  MoveL 4062 to (-40.22, 47.43, 69.25) mm, rotated rx 180 ry 0 rz -180 deg; joints [-39.002, -24.615, 92.109, 64.701, 44.116, -56.64]
  Call Extruder(62.49416)
  MoveL 4063 to (-40.17, 47.23, 69.25) mm, rotated rx 180 ry 0 rz 180 deg; joints [-38.962, -24.627, 92.115, 64.664, 44.084, -56.61]
  MoveL 4064 to (-40.17, 47.23, 69.25) mm, rotated rx 180 ry 0 rz 180 deg; joints [-38.962, -24.627, 92.115, 64.664, 44.084, -56.61]
  Call Extruder(62.60834)
  MoveL 4065 to (-40.13, 47.02, 69.25) mm, rotated rx 180 ry 0 rz 180 deg; joints [-38.921, -24.64, 92.122, 64.627, 44.053, -56.579]
  MoveL 4066 to (-40.13, 47.02, 69.25) mm, rotated rx 180 ry 0 rz 180 deg; joints [-38.921, -24.64, 92.122, 64.627, 44.053, -56.579]
  Call Extruder(62.72297)
  MoveL 4067 to (-40.08, 46.82, 69.25) mm, rotated rx 180 ry 0 rz -180 deg; joints [-38.88, -24.652, 92.129, 64.589, 44.021, -56.549]
  MoveL 4068 to (-40.08, 46.82, 69.25) mm, rotated rx 180 ry 0 rz -180 deg; joints [-38.88, -24.652, 92.129, 64.589, 44.021, -56.549]
  Call Extruder(62.83806)
  MoveL 4069 to (-40.04, 46.61, 69.25) mm, rotated rx 180 ry 0 rz 180 deg; joints [-38.839, -24.664, 92.136, 64.552, 43.989, -56.519]
  MoveL 4070 to (-40.04, 46.61, 69.25) mm, rotated rx 180 ry 0 rz 180 deg; joints [-38.839, -24.664, 92.136, 64.552, 43.989, -56.519]
  Call Extruder(62.96029)
  MoveL 4071 to (-39.98, 46.4, 69.25) mm, rotated rx 180 ry 0 rz 180 deg; joints [-38.795, -24.676, 92.142, 64.512, 43.955, -56.487]
  MoveL 4072 to (-39.98, 46.4, 69.25) mm, rotated rx 180 ry 0 rz 180 deg; joints [-38.795, -24.676, 92.142, 64.512, 43.955, -56.487]
  Call Extruder(63.08996)
  MoveL 4073 to (-39.92, 46.18, 69.25) mm, rotated rx 180 ry 0 rz -180 deg; joints [-38.748, -24.687, 92.148, 64.469, 43.917, -56.453]
  MoveL 4074 to (-39.92, 46.18, 69.25) mm, rotated rx 180 ry 0 rz -180 deg; joints [-38.748, -24.687, 92.148, 64.469, 43.917, -56.453]
  Call Extruder(63.22019)
  MoveL 4075 to (-39.85, 45.95, 69.25) mm, rotated rx 180 ry 0 rz 180 deg; joints [-38.7, -24.699, 92.155, 64.427, 43.88, -56.419]
  MoveL 4076 to (-39.85, 45.95, 69.25) mm, rotated rx 180 ry 0 rz 180 deg; joints [-38.7, -24.699, 92.155, 64.427, 43.88, -56.419]
  Call Extruder(63.35098)
  MoveL 4077 to (-39.78, 45.73, 69.25) mm, rotated rx 180 ry 0 rz 180 deg; joints [-38.653, -24.71, 92.161, 64.384, 43.843, -56.385]
  MoveL 4078 to (-39.78, 45.73, 69.25) mm, rotated rx 180 ry 0 rz 180 deg; joints [-38.653, -24.71, 92.161, 64.384, 43.843, -56.385]
  Call Extruder(63.48234)
  MoveL 4079 to (-39.71, 45.51, 69.25) mm, rotated rx 180 ry 0 rz 180 deg; joints [-38.605, -24.721, 92.167, 64.341, 43.805, -56.351]
  MoveL 4080 to (-39.71, 45.51, 69.25) mm, rotated rx 180 ry 0 rz 180 deg; joints [-38.605, -24.721, 92.167, 64.341, 43.805, -56.351]
  Call Extruder(63.59424)
  MoveL 4081 to (-39.65, 45.32, 69.25) mm, rotated rx -180 ry 0 rz 180 deg; joints [-38.565, -24.73, 92.172, 64.305, 43.774, -56.322]
  MoveL 4082 to (-39.65, 45.32, 69.25) mm, rotated rx -180 ry 0 rz 180 deg; joints [-38.565, -24.73, 92.172, 64.305, 43.774, -56.322]
  Call Extruder(63.70659)
  MoveL 4083 to (-39.59, 45.13, 69.25) mm, rotated rx 180 ry 0 rz 180 deg; joints [-38.524, -24.74, 92.177, 64.268, 43.741, -56.293]
  MoveL 4084 to (-39.59, 45.13, 69.25) mm, rotated rx 180 ry 0 rz 180 deg; joints [-38.524, -24.74, 92.177, 64.268, 43.741, -56.293]
  Call Extruder(63.81938)
  MoveL 4085 to (-39.53, 44.94, 69.25) mm, rotated rx 180 ry 0 rz -180 deg; joints [-38.483, -24.749, 92.182, 64.232, 43.709, -56.264]
  MoveL 4086 to (-39.53, 44.94, 69.25) mm, rotated rx 180 ry 0 rz -180 deg; joints [-38.483, -24.749, 92.182, 64.232, 43.709, -56.264]
  Call Extruder(63.93261)
  MoveL 4087 to (-39.47, 44.75, 69.25) mm, rotated rx -180 ry 0 rz 180 deg; joints [-38.443, -24.758, 92.187, 64.195, 43.677, -56.235]
  MoveL 4088 to (-39.47, 44.75, 69.25) mm, rotated rx -180 ry 0 rz 180 deg; joints [-38.443, -24.758, 92.187, 64.195, 43.677, -56.235]
  Call Extruder(64.04629)
  MoveL 4089 to (-39.41, 44.56, 69.25) mm, rotated rx -180 ry 0 rz 180 deg; joints [-38.402, -24.767, 92.192, 64.159, 43.645, -56.206]
  MoveL 4090 to (-39.41, 44.56, 69.25) mm, rotated rx -180 ry 0 rz 180 deg; joints [-38.402, -24.767, 92.192, 64.159, 43.645, -56.206]
  Call Extruder(64.22825)
  MoveL 4091 to (-39.29, 44.27, 69.25) mm, rotated rx 180 ry 0 rz 180 deg; joints [-38.335, -24.778, 92.198, 64.1, 43.592, -56.161]
  MoveL 4092 to (-39.29, 44.27, 69.25) mm, rotated rx 180 ry 0 rz 180 deg; joints [-38.335, -24.778, 92.198, 64.1, 43.592, -56.161]
  Call Extruder(64.41097)
  MoveL 4093 to (-39.16, 43.98, 69.25) mm, rotated rx -180 ry 0 rz 180 deg; joints [-38.269, -24.789, 92.204, 64.042, 43.539, -56.115]
  MoveL 4094 to (-39.16, 43.98, 69.25) mm, rotated rx -180 ry 0 rz 180 deg; joints [-38.269, -24.789, 92.204, 64.042, 43.539, -56.115]
  Call Extruder(64.58138)
  MoveL 4095 to (-39.05, 43.71, 69.25) mm, rotated rx 180 ry 0 rz 180 deg; joints [-38.207, -24.799, 92.21, 63.987, 43.49, -56.073]
  MoveL 4096 to (-39.05, 43.71, 69.25) mm, rotated rx 180 ry 0 rz 180 deg; joints [-38.207, -24.799, 92.21, 63.987, 43.49, -56.073]
  Call Extruder(64.73937)
  MoveL 4097 to (-38.94, 43.46, 69.25) mm, rotated rx 180 ry 0 rz 180 deg; joints [-38.149, -24.808, 92.215, 63.936, 43.444, -56.034]
  MoveL 4098 to (-38.94, 43.46, 69.25) mm, rotated rx 180 ry 0 rz 180 deg; joints [-38.149, -24.808, 92.215, 63.936, 43.444, -56.034]
  Call Extruder(64.89795)
  MoveL 4099 to (-38.84, 43.21, 69.25) mm, rotated rx 180 ry 0 rz 180 deg; joints [-38.092, -24.818, 92.22, 63.886, 43.398, -55.994]
  MoveL 4100 to (-38.84, 43.21, 69.25) mm, rotated rx 180 ry 0 rz 180 deg; joints [-38.092, -24.818, 92.22, 63.886, 43.398, -55.994]
  Call Extruder(65.10412)
  MoveL 4101 to (-38.66, 42.91, 69.25) mm, rotated rx 180 ry 0 rz 180 deg; joints [-38.016, -24.824, 92.224, 63.821, 43.336, -55.945]
  MoveL 4102 to (-38.66, 42.91, 69.25) mm, rotated rx 180 ry 0 rz 180 deg; joints [-38.016, -24.824, 92.224, 63.821, 43.336, -55.945]
  Call Extruder(65.31106)
  MoveL 4103 to (-38.49, 42.6, 69.25) mm, rotated rx 180 ry 0 rz -180 deg; joints [-37.939, -24.83, 92.227, 63.756, 43.274, -55.896]
  MoveL 4104 to (-38.49, 42.6, 69.25) mm, rotated rx 180 ry 0 rz -180 deg; joints [-37.939, -24.83, 92.227, 63.756, 43.274, -55.896]
  Call Extruder(65.51879)
  MoveL 4105 to (-38.31, 42.3, 69.25) mm, rotated rx -180 ry 0 rz 180 deg; joints [-37.863, -24.837, 92.23, 63.69, 43.212, -55.847]
  MoveL 4106 to (-38.31, 42.3, 69.25) mm, rotated rx -180 ry 0 rz 180 deg; joints [-37.863, -24.837, 92.23, 63.69, 43.212, -55.847]
  Call Extruder(65.72729)
  MoveL 4107 to (-38.14, 41.99, 69.25) mm, rotated rx 180 ry 0 rz 180 deg; joints [-37.787, -24.843, 92.234, 63.625, 43.15, -55.797]
  MoveL 4108 to (-38.14, 41.99, 69.25) mm, rotated rx 180 ry 0 rz 180 deg; joints [-37.787, -24.843, 92.234, 63.625, 43.15, -55.797]
  Call Extruder(65.90684)
  MoveL 4109 to (-37.96, 41.75, 69.25) mm, rotated rx -180 ry 0 rz 180 deg; joints [-37.72, -24.844, 92.235, 63.57, 43.096, -55.757]
  MoveL 4110 to (-37.96, 41.75, 69.25) mm, rotated rx -180 ry 0 rz 180 deg; joints [-37.72, -24.844, 92.235, 63.57, 43.096, -55.757]
  Call Extruder(66.24028)
  MoveL 4111 to (-37.63, 41.3, 69.25) mm, rotated rx 180 ry 0 rz -180 deg; joints [-37.598, -24.846, 92.236, 63.468, 42.995, -55.682]
  MoveL 4112 to (-37.63, 41.3, 69.25) mm, rotated rx 180 ry 0 rz -180 deg; joints [-37.598, -24.846, 92.236, 63.468, 42.995, -55.682]
  Call Extruder(66.57490)
  MoveL 4113 to (-37.3, 40.85, 69.25) mm, rotated rx 180 ry 0 rz 180 deg; joints [-37.475, -24.848, 92.237, 63.366, 42.894, -55.606]
  Call Extruder(67.40283)
  MoveL 4114 to (-36.39, 39.81, 69.25) mm, rotated rx -180 ry 0 rz 180 deg; joints [-37.173, -24.836, 92.23, 63.119, 42.642, -55.429]
  Call Extruder(68.23074)
  MoveL 4115 to (-35.35, 38.9, 69.25) mm, rotated rx 180 ry 0 rz 180 deg; joints [-36.876, -24.799, 92.21, 62.885, 42.391, -55.266]
  Call Extruder(68.39804)
  MoveL 4116 to (-35.13, 38.73, 69.25) mm, rotated rx -180 ry 0 rz -180 deg; joints [-36.818, -24.789, 92.204, 62.84, 42.34, -55.236]
  MoveL 4117 to (-35.13, 38.73, 69.25) mm, rotated rx -180 ry 0 rz -180 deg; joints [-36.818, -24.789, 92.204, 62.84, 42.34, -55.236]
  Call Extruder(68.73147)
  MoveL 4118 to (-34.68, 38.41, 69.25) mm, rotated rx 180 ry 0 rz 180 deg; joints [-36.701, -24.767, 92.192, 62.751, 42.24, -55.176]
  MoveL 4119 to (-34.68, 38.41, 69.25) mm, rotated rx 180 ry 0 rz 180 deg; joints [-36.701, -24.767, 92.192, 62.751, 42.24, -55.176]
  Call Extruder(69.06371)
  MoveL 4120 to (-34.23, 38.08, 69.25) mm, rotated rx 180 ry 0 rz -180 deg; joints [-36.584, -24.745, 92.18, 62.661, 42.14, -55.115]
  MoveL 4121 to (-34.23, 38.08, 69.25) mm, rotated rx 180 ry 0 rz -180 deg; joints [-36.584, -24.745, 92.18, 62.661, 42.14, -55.115]
  Call Extruder(69.18141)
  MoveL 4122 to (-34.05, 37.98, 69.25) mm, rotated rx 180 ry 0 rz 180 deg; joints [-36.544, -24.735, 92.175, 62.632, 42.105, -55.096]
  MoveL 4123 to (-34.05, 37.98, 69.25) mm, rotated rx 180 ry 0 rz 180 deg; joints [-36.544, -24.735, 92.175, 62.632, 42.105, -55.096]
  Call Extruder(69.38913)
  MoveL 4124 to (-33.75, 37.8, 69.25) mm, rotated rx 180 ry 0 rz 180 deg; joints [-36.474, -24.717, 92.165, 62.58, 42.043, -55.062]
  MoveL 4125 to (-33.75, 37.8, 69.25) mm, rotated rx 180 ry 0 rz 180 deg; joints [-36.474, -24.717, 92.165, 62.58, 42.043, -55.062]
  Call Extruder(69.59607)
  MoveL 4126 to (-33.45, 37.63, 69.25) mm, rotated rx 180 ry 0 rz 180 deg; joints [-36.403, -24.699, 92.155, 62.527, 41.982, -55.028]
  MoveL 4127 to (-33.45, 37.63, 69.25) mm, rotated rx 180 ry 0 rz 180 deg; joints [-36.403, -24.699, 92.155, 62.527, 41.982, -55.028]
  Call Extruder(69.80224)
  MoveL 4128 to (-33.14, 37.45, 69.25) mm, rotated rx 180 ry 0 rz 180 deg; joints [-36.333, -24.68, 92.144, 62.475, 41.921, -54.994]
  MoveL 4129 to (-33.14, 37.45, 69.25) mm, rotated rx 180 ry 0 rz 180 deg; joints [-36.333, -24.68, 92.144, 62.475, 41.921, -54.994]
  Call Extruder(69.98392)
  MoveL 4130 to (-32.86, 37.31, 69.25) mm, rotated rx 180 ry 0 rz 180 deg; joints [-36.272, -24.662, 92.134, 62.431, 41.867, -54.966]
  MoveL 4131 to (-32.86, 37.31, 69.25) mm, rotated rx 180 ry 0 rz 180 deg; joints [-36.272, -24.662, 92.134, 62.431, 41.867, -54.966]
  Call Extruder(70.14192)
  MoveL 4132 to (-32.62, 37.2, 69.25) mm, rotated rx 180 ry 0 rz 180 deg; joints [-36.221, -24.644, 92.124, 62.395, 41.822, -54.944]
  MoveL 4133 to (-32.62, 37.2, 69.25) mm, rotated rx 180 ry 0 rz 180 deg; joints [-36.221, -24.644, 92.124, 62.395, 41.822, -54.944]
  Call Extruder(70.29931)
  MoveL 4134 to (-32.37, 37.1, 69.25) mm, rotated rx 180 ry 0 rz 180 deg; joints [-36.17, -24.626, 92.115, 62.359, 41.776, -54.922]
  MoveL 4135 to (-32.37, 37.1, 69.25) mm, rotated rx 180 ry 0 rz 180 deg; joints [-36.17, -24.626, 92.115, 62.359, 41.776, -54.922]
  Call Extruder(70.48203)
  MoveL 4136 to (-32.08, 36.97, 69.25) mm, rotated rx 180 ry 0 rz 180 deg; joints [-36.112, -24.604, 92.103, 62.318, 41.724, -54.897]
  MoveL 4137 to (-32.08, 36.97, 69.25) mm, rotated rx 180 ry 0 rz 180 deg; joints [-36.112, -24.604, 92.103, 62.318, 41.724, -54.897]
  Call Extruder(70.66398)
  MoveL 4138 to (-31.78, 36.85, 69.25) mm, rotated rx 180 ry 0 rz 180 deg; joints [-36.053, -24.583, 92.091, 62.277, 41.671, -54.872]
  MoveL 4139 to (-31.78, 36.85, 69.25) mm, rotated rx 180 ry 0 rz 180 deg; joints [-36.053, -24.583, 92.091, 62.277, 41.671, -54.872]
  Call Extruder(70.81131)
  MoveL 4140 to (-31.54, 36.76, 69.25) mm, rotated rx -180 ry 0 rz 180 deg; joints [-36.006, -24.565, 92.081, 62.245, 41.629, -54.853]
  MoveL 4141 to (-31.54, 36.76, 69.25) mm, rotated rx -180 ry 0 rz 180 deg; joints [-36.006, -24.565, 92.081, 62.245, 41.629, -54.853]
  Call Extruder(70.92455)
  MoveL 4142 to (-31.35, 36.7, 69.25) mm, rotated rx 180 ry 0 rz 180 deg; joints [-35.971, -24.549, 92.072, 62.221, 41.597, -54.839]
  MoveL 4143 to (-31.35, 36.7, 69.25) mm, rotated rx 180 ry 0 rz 180 deg; joints [-35.971, -24.549, 92.072, 62.221, 41.597, -54.839]
  Call Extruder(71.03734)
  MoveL 4144 to (-31.17, 36.64, 69.25) mm, rotated rx 180 ry 0 rz 180 deg; joints [-35.936, -24.534, 92.064, 62.198, 41.565, -54.826]
  MoveL 4145 to (-31.17, 36.64, 69.25) mm, rotated rx 180 ry 0 rz 180 deg; joints [-35.936, -24.534, 92.064, 62.198, 41.565, -54.826]
  Call Extruder(71.14968)
  MoveL 4146 to (-30.98, 36.58, 69.25) mm, rotated rx 180 ry 0 rz 180 deg; joints [-35.901, -24.519, 92.055, 62.174, 41.534, -54.812]
  MoveL 4147 to (-30.98, 36.58, 69.25) mm, rotated rx 180 ry 0 rz 180 deg; joints [-35.901, -24.519, 92.055, 62.174, 41.534, -54.812]
  Call Extruder(71.26159)
  MoveL 4148 to (-30.79, 36.52, 69.25) mm, rotated rx 180 ry 0 rz 180 deg; joints [-35.867, -24.504, 92.047, 62.151, 41.502, -54.799]
  MoveL 4149 to (-30.79, 36.52, 69.25) mm, rotated rx 180 ry 0 rz 180 deg; joints [-35.867, -24.504, 92.047, 62.151, 41.502, -54.799]
  Call Extruder(71.38299)
  MoveL 4150 to (-30.58, 36.45, 69.25) mm, rotated rx 180 ry 0 rz 180 deg; joints [-35.829, -24.487, 92.037, 62.125, 41.468, -54.784]
  MoveL 4151 to (-30.58, 36.45, 69.25) mm, rotated rx 180 ry 0 rz 180 deg; joints [-35.829, -24.487, 92.037, 62.125, 41.468, -54.784]
  Call Extruder(71.51378)
  MoveL 4152 to (-30.36, 36.39, 69.25) mm, rotated rx 180 ry 0 rz 180 deg; joints [-35.788, -24.468, 92.027, 62.098, 41.431, -54.769]
  MoveL 4153 to (-30.36, 36.39, 69.25) mm, rotated rx 180 ry 0 rz 180 deg; joints [-35.788, -24.468, 92.027, 62.098, 41.431, -54.769]
  Call Extruder(71.64400)
  MoveL 4154 to (-30.14, 36.32, 69.25) mm, rotated rx 180 ry 0 rz 180 deg; joints [-35.748, -24.45, 92.017, 62.072, 41.394, -54.753]
  MoveL 4155 to (-30.14, 36.32, 69.25) mm, rotated rx 180 ry 0 rz 180 deg; joints [-35.748, -24.45, 92.017, 62.072, 41.394, -54.753]
  Call Extruder(71.77367)
  MoveL 4156 to (-29.91, 36.25, 69.25) mm, rotated rx -180 ry 0 rz 180 deg; joints [-35.708, -24.431, 92.006, 62.045, 41.358, -54.738]
  MoveL 4157 to (-29.91, 36.25, 69.25) mm, rotated rx -180 ry 0 rz 180 deg; joints [-35.708, -24.431, 92.006, 62.045, 41.358, -54.738]
  Call Extruder(71.90276)
  MoveL 4158 to (-29.69, 36.18, 69.25) mm, rotated rx 180 ry 0 rz 180 deg; joints [-35.668, -24.412, 91.996, 62.018, 41.321, -54.723]
  MoveL 4159 to (-29.69, 36.18, 69.25) mm, rotated rx 180 ry 0 rz 180 deg; joints [-35.668, -24.412, 91.996, 62.018, 41.321, -54.723]
  Call Extruder(72.01784)
  MoveL 4160 to (-29.48, 36.14, 69.25) mm, rotated rx 180 ry 0 rz 180 deg; joints [-35.634, -24.394, 91.986, 61.997, 41.29, -54.711]
  MoveL 4161 to (-29.48, 36.14, 69.25) mm, rotated rx 180 ry 0 rz 180 deg; joints [-35.634, -24.394, 91.986, 61.997, 41.29, -54.711]
  Call Extruder(72.13246)
  MoveL 4162 to (-29.28, 36.09, 69.25) mm, rotated rx -180 ry 0 rz 180 deg; joints [-35.601, -24.376, 91.976, 61.975, 41.258, -54.7]
  MoveL 4163 to (-29.28, 36.09, 69.25) mm, rotated rx -180 ry 0 rz 180 deg; joints [-35.601, -24.376, 91.976, 61.975, 41.258, -54.7]
  Call Extruder(72.24663)
  MoveL 4164 to (-29.08, 36.05, 69.25) mm, rotated rx 180 ry 0 rz 180 deg; joints [-35.567, -24.357, 91.965, 61.954, 41.227, -54.689]
  MoveL 4165 to (-29.08, 36.05, 69.25) mm, rotated rx 180 ry 0 rz 180 deg; joints [-35.567, -24.357, 91.965, 61.954, 41.227, -54.689]
  Call Extruder(72.36034)
  MoveL 4166 to (-28.87, 36, 69.25) mm, rotated rx 180 ry 0 rz 180 deg; joints [-35.533, -24.339, 91.955, 61.933, 41.196, -54.678]
  MoveL 4167 to (-28.87, 36, 69.25) mm, rotated rx 180 ry 0 rz 180 deg; joints [-35.533, -24.339, 91.955, 61.933, 41.196, -54.678]
  Call Extruder(72.48576)
  MoveL 4168 to (-28.65, 35.96, 69.25) mm, rotated rx 180 ry 0 rz 180 deg; joints [-35.497, -24.318, 91.944, 61.91, 41.162, -54.665]
  MoveL 4169 to (-28.65, 35.96, 69.25) mm, rotated rx 180 ry 0 rz 180 deg; joints [-35.497, -24.318, 91.944, 61.91, 41.162, -54.665]
  Call Extruder(72.62274)
  MoveL 4170 to (-28.4, 35.91, 69.25) mm, rotated rx 180 ry 0 rz 180 deg; joints [-35.457, -24.296, 91.931, 61.885, 41.124, -54.652]
  MoveL 4171 to (-28.4, 35.91, 69.25) mm, rotated rx 180 ry 0 rz 180 deg; joints [-35.457, -24.296, 91.931, 61.885, 41.124, -54.652]
  Call Extruder(72.75911)
  MoveL 4172 to (-28.15, 35.86, 69.25) mm, rotated rx -180 ry 0 rz 180 deg; joints [-35.417, -24.273, 91.918, 61.86, 41.087, -54.64]
  MoveL 4173 to (-28.15, 35.86, 69.25) mm, rotated rx -180 ry 0 rz 180 deg; joints [-35.417, -24.273, 91.918, 61.86, 41.087, -54.64]
  Call Extruder(72.89487)
  MoveL 4174 to (-27.9, 35.81, 69.25) mm, rotated rx 180 ry 0 rz 180 deg; joints [-35.377, -24.25, 91.905, 61.835, 41.05, -54.626]
  MoveL 4175 to (-27.9, 35.81, 69.25) mm, rotated rx 180 ry 0 rz 180 deg; joints [-35.377, -24.25, 91.905, 61.835, 41.05, -54.626]
  Call Extruder(73.03001)
  MoveL 4176 to (-27.65, 35.76, 69.25) mm, rotated rx -180 ry 0 rz 180 deg; joints [-35.337, -24.227, 91.893, 61.81, 41.012, -54.614]
  MoveL 4177 to (-27.65, 35.76, 69.25) mm, rotated rx -180 ry 0 rz 180 deg; joints [-35.337, -24.227, 91.893, 61.81, 41.012, -54.614]
  Call Extruder(73.16455)
  MoveL 4178 to (-27.4, 35.71, 69.25) mm, rotated rx -180 ry 0 rz 180 deg; joints [-35.297, -24.204, 91.88, 61.785, 40.975, -54.601]
  MoveL 4179 to (-27.4, 35.71, 69.25) mm, rotated rx -180 ry 0 rz 180 deg; joints [-35.297, -24.204, 91.88, 61.785, 40.975, -54.601]
  Call Extruder(73.29848)
  MoveL 4180 to (-27.15, 35.66, 69.25) mm, rotated rx 180 ry 0 rz 180 deg; joints [-35.258, -24.181, 91.867, 61.76, 40.938, -54.588]
  MoveL 4181 to (-27.15, 35.66, 69.25) mm, rotated rx 180 ry 0 rz 180 deg; joints [-35.258, -24.181, 91.867, 61.76, 40.938, -54.588]
  Call Extruder(73.44634)
  MoveL 4182 to (-26.87, 35.61, 69.25) mm, rotated rx 180 ry 0 rz 180 deg; joints [-35.215, -24.155, 91.852, 61.734, 40.898, -54.574]
  MoveL 4183 to (-26.87, 35.61, 69.25) mm, rotated rx 180 ry 0 rz 180 deg; joints [-35.215, -24.155, 91.852, 61.734, 40.898, -54.574]
  Call Extruder(73.60807)
  MoveL 4184 to (-26.57, 35.56, 69.25) mm, rotated rx 180 ry 0 rz 180 deg; joints [-35.168, -24.126, 91.836, 61.705, 40.854, -54.56]
  MoveL 4185 to (-26.57, 35.56, 69.25) mm, rotated rx 180 ry 0 rz 180 deg; joints [-35.168, -24.126, 91.836, 61.705, 40.854, -54.56]
  Call Extruder(73.76908)
  MoveL 4186 to (-26.26, 35.51, 69.25) mm, rotated rx 180 ry 0 rz -180 deg; joints [-35.122, -24.097, 91.82, 61.677, 40.81, -54.546]
  MoveL 4187 to (-26.26, 35.51, 69.25) mm, rotated rx 180 ry 0 rz -180 deg; joints [-35.122, -24.097, 91.82, 61.677, 40.81, -54.546]
  Call Extruder(73.92935)
  MoveL 4188 to (-25.96, 35.47, 69.25) mm, rotated rx 180 ry 0 rz 180 deg; joints [-35.075, -24.068, 91.803, 61.649, 40.766, -54.532]
  MoveL 4189 to (-25.96, 35.47, 69.25) mm, rotated rx 180 ry 0 rz 180 deg; joints [-35.075, -24.068, 91.803, 61.649, 40.766, -54.532]
  Call Extruder(74.08890)
  MoveL 4190 to (-25.65, 35.42, 69.25) mm, rotated rx 180 ry 0 rz 180 deg; joints [-35.029, -24.039, 91.787, 61.621, 40.723, -54.518]
  MoveL 4191 to (-25.65, 35.42, 69.25) mm, rotated rx 180 ry 0 rz 180 deg; joints [-35.029, -24.039, 91.787, 61.621, 40.723, -54.518]
  Call Extruder(74.24773)
  MoveL 4192 to (-25.34, 35.37, 69.25) mm, rotated rx 180 ry 0 rz -180 deg; joints [-34.983, -24.009, 91.77, 61.593, 40.679, -54.504]
  MoveL 4193 to (-25.34, 35.37, 69.25) mm, rotated rx 180 ry 0 rz -180 deg; joints [-34.983, -24.009, 91.77, 61.593, 40.679, -54.504]
  Call Extruder(74.42640)
  MoveL 4194 to (-25, 35.32, 69.25) mm, rotated rx 180 ry 0 rz -180 deg; joints [-34.932, -23.976, 91.751, 61.563, 40.631, -54.49]
  MoveL 4195 to (-25, 35.32, 69.25) mm, rotated rx 180 ry 0 rz -180 deg; joints [-34.932, -23.976, 91.751, 61.563, 40.631, -54.49]
  Call Extruder(74.62484)
  MoveL 4196 to (-24.61, 35.27, 69.25) mm, rotated rx 180 ry 0 rz 180 deg; joints [-34.877, -23.937, 91.73, 61.53, 40.577, -54.475]
  MoveL 4197 to (-24.61, 35.27, 69.25) mm, rotated rx 180 ry 0 rz 180 deg; joints [-34.877, -23.937, 91.73, 61.53, 40.577, -54.475]
  Call Extruder(74.82241)
  MoveL 4198 to (-24.22, 35.23, 69.25) mm, rotated rx 180 ry 0 rz -180 deg; joints [-34.821, -23.899, 91.708, 61.498, 40.524, -54.46]
  MoveL 4199 to (-24.22, 35.23, 69.25) mm, rotated rx 180 ry 0 rz -180 deg; joints [-34.821, -23.899, 91.708, 61.498, 40.524, -54.46]
  Call Extruder(75.01912)
  MoveL 4200 to (-23.84, 35.18, 69.25) mm, rotated rx 180 ry 0 rz -180 deg; joints [-34.766, -23.861, 91.686, 61.465, 40.471, -54.444]
  MoveL 4201 to (-23.84, 35.18, 69.25) mm, rotated rx 180 ry 0 rz -180 deg; joints [-34.766, -23.861, 91.686, 61.465, 40.471, -54.444]
  Call Extruder(75.21496)
  MoveL 4202 to (-23.45, 35.14, 69.25) mm, rotated rx 180 ry 0 rz 180 deg; joints [-34.711, -23.822, 91.664, 61.433, 40.419, -54.429]
  MoveL 4203 to (-23.45, 35.14, 69.25) mm, rotated rx 180 ry 0 rz 180 deg; joints [-34.711, -23.822, 91.664, 61.433, 40.419, -54.429]
  Call Extruder(75.51035)
  MoveL 4204 to (-22.86, 35.09, 69.25) mm, rotated rx 180 ry 0 rz 180 deg; joints [-34.631, -23.762, 91.63, 61.389, 40.342, -54.41]
  MoveL 4205 to (-22.86, 35.09, 69.25) mm, rotated rx 180 ry 0 rz 180 deg; joints [-34.631, -23.762, 91.63, 61.389, 40.342, -54.41]
  Call Extruder(75.80442)
  MoveL 4206 to (-22.27, 35.05, 69.25) mm, rotated rx -180 ry 0 rz 180 deg; joints [-34.552, -23.702, 91.596, 61.344, 40.265, -54.391]
  MoveL 4207 to (-22.27, 35.05, 69.25) mm, rotated rx -180 ry 0 rz 180 deg; joints [-34.552, -23.702, 91.596, 61.344, 40.265, -54.391]
  Call Extruder(76.09715)
  MoveL 4208 to (-21.68, 35, 69.25) mm, rotated rx 180 ry 0 rz 180 deg; joints [-34.473, -23.641, 91.561, 61.3, 40.188, -54.372]
  MoveL 4209 to (-21.68, 35, 69.25) mm, rotated rx 180 ry 0 rz 180 deg; joints [-34.473, -23.641, 91.561, 61.3, 40.188, -54.372]
  Call Extruder(76.67060)
  MoveL 4210 to (-20.52, 34.95, 69.25) mm, rotated rx 180 ry 0 rz 180 deg; joints [-34.326, -23.518, 91.491, 61.221, 40.043, -54.341]
  MoveL 4211 to (-20.52, 34.95, 69.25) mm, rotated rx 180 ry 0 rz 180 deg; joints [-34.326, -23.518, 91.491, 61.221, 40.043, -54.341]
  Call Extruder(77.38456)
  MoveL 4212 to (-19.06, 34.91, 69.25) mm, rotated rx 180 ry 0 rz 180 deg; joints [-34.146, -23.363, 91.402, 61.127, 39.865, -54.307]
  Call Extruder(194.23128)
  MoveL 4213 to (219.06, 34.91, 69.25) mm, rotated rx -180 ry 0 rz 180 deg; joints [-18.248, 8.607, 63.654, 47.26, 25.237, -44.389]
  Call Extruder(194.65984)
  MoveL 4214 to (219.94, 34.93, 69.25) mm, rotated rx 180 ry 0 rz 180 deg; joints [-18.218, 8.753, 63.486, 47.175, 25.231, -44.304]
  MoveL 4215 to (219.94, 34.93, 69.25) mm, rotated rx 180 ry 0 rz 180 deg; joints [-18.218, 8.753, 63.486, 47.175, 25.231, -44.304]
  Call Extruder(195.23329)
  MoveL 4216 to (221.1, 34.97, 69.25) mm, rotated rx 180 ry 0 rz 180 deg; joints [-18.181, 8.948, 63.26, 47.064, 25.226, -44.195]
  MoveL 4217 to (221.1, 34.97, 69.25) mm, rotated rx 180 ry 0 rz 180 deg; joints [-18.181, 8.948, 63.26, 47.064, 25.226, -44.195]
  Call Extruder(195.66760)
  MoveL 4218 to (221.97, 35.02, 69.25) mm, rotated rx 180 ry 0 rz 180 deg; joints [-18.154, 9.097, 63.088, 46.982, 25.223, -44.113]
  MoveL 4219 to (221.97, 35.02, 69.25) mm, rotated rx 180 ry 0 rz 180 deg; joints [-18.154, 9.097, 63.088, 46.982, 25.223, -44.113]
  Call Extruder(195.96166)
  MoveL 4220 to (222.56, 35.07, 69.25) mm, rotated rx 180 ry 0 rz 180 deg; joints [-18.138, 9.197, 62.971, 46.929, 25.223, -44.061]
  MoveL 4221 to (222.56, 35.07, 69.25) mm, rotated rx 180 ry 0 rz 180 deg; joints [-18.138, 9.197, 62.971, 46.929, 25.223, -44.061]
  Call Extruder(196.25705)
  MoveL 4222 to (223.15, 35.11, 69.25) mm, rotated rx 180 ry 0 rz -180 deg; joints [-18.121, 9.298, 62.853, 46.876, 25.223, -44.007]
  MoveL 4223 to (223.15, 35.11, 69.25) mm, rotated rx 180 ry 0 rz -180 deg; joints [-18.121, 9.298, 62.853, 46.876, 25.223, -44.007]
  Call Extruder(196.50328)
  MoveL 4224 to (223.64, 35.16, 69.25) mm, rotated rx -180 ry 0 rz -180 deg; joints [-18.109, 9.383, 62.755, 46.833, 25.224, -43.964]
  MoveL 4225 to (223.64, 35.16, 69.25) mm, rotated rx -180 ry 0 rz -180 deg; joints [-18.109, 9.383, 62.755, 46.833, 25.224, -43.964]
  Call Extruder(196.69999)
  MoveL 4226 to (224.03, 35.21, 69.25) mm, rotated rx -180 ry 0 rz 180 deg; joints [-18.1, 9.45, 62.676, 46.801, 25.225, -43.931]
  MoveL 4227 to (224.03, 35.21, 69.25) mm, rotated rx -180 ry 0 rz 180 deg; joints [-18.1, 9.45, 62.676, 46.801, 25.225, -43.931]
  Call Extruder(196.89757)
  MoveL 4228 to (224.42, 35.25, 69.25) mm, rotated rx 180 ry 0 rz 180 deg; joints [-18.091, 9.518, 62.597, 46.768, 25.227, -43.898]
  MoveL 4229 to (224.42, 35.25, 69.25) mm, rotated rx 180 ry 0 rz 180 deg; joints [-18.091, 9.518, 62.597, 46.768, 25.227, -43.898]
  Call Extruder(197.09601)
  MoveL 4230 to (224.8, 35.3, 69.25) mm, rotated rx 180 ry 0 rz 180 deg; joints [-18.082, 9.585, 62.518, 46.736, 25.229, -43.865]
  MoveL 4231 to (224.8, 35.3, 69.25) mm, rotated rx 180 ry 0 rz 180 deg; joints [-18.082, 9.585, 62.518, 46.736, 25.229, -43.865]
  Call Extruder(197.29532)
  MoveL 4232 to (225.19, 35.34, 69.25) mm, rotated rx 180 ry 0 rz 180 deg; joints [-18.073, 9.653, 62.439, 46.703, 25.23, -43.832]
  MoveL 4233 to (225.19, 35.34, 69.25) mm, rotated rx 180 ry 0 rz 180 deg; joints [-18.073, 9.653, 62.439, 46.703, 25.23, -43.832]
  Call Extruder(197.45414)
  MoveL 4234 to (225.5, 35.39, 69.25) mm, rotated rx -180 ry 0 rz 180 deg; joints [-18.068, 9.707, 62.376, 46.679, 25.233, -43.807]
  MoveL 4235 to (225.5, 35.39, 69.25) mm, rotated rx -180 ry 0 rz 180 deg; joints [-18.068, 9.707, 62.376, 46.679, 25.233, -43.807]
  Call Extruder(197.61369)
  MoveL 4236 to (225.8, 35.44, 69.25) mm, rotated rx 180 ry 0 rz 180 deg; joints [-18.062, 9.761, 62.312, 46.655, 25.235, -43.783]
  MoveL 4237 to (225.8, 35.44, 69.25) mm, rotated rx 180 ry 0 rz 180 deg; joints [-18.062, 9.761, 62.312, 46.655, 25.235, -43.783]
  Call Extruder(197.77397)
  MoveL 4238 to (226.11, 35.49, 69.25) mm, rotated rx 180 ry 0 rz 180 deg; joints [-18.056, 9.815, 62.249, 46.631, 25.238, -43.758]
  MoveL 4239 to (226.11, 35.49, 69.25) mm, rotated rx 180 ry 0 rz 180 deg; joints [-18.056, 9.815, 62.249, 46.631, 25.238, -43.758]
  Call Extruder(197.93497)
  MoveL 4240 to (226.41, 35.54, 69.25) mm, rotated rx -180 ry 0 rz 180 deg; joints [-18.051, 9.87, 62.185, 46.607, 25.24, -43.733]
  MoveL 4241 to (226.41, 35.54, 69.25) mm, rotated rx -180 ry 0 rz 180 deg; joints [-18.051, 9.87, 62.185, 46.607, 25.24, -43.733]
  Call Extruder(198.09670)
  MoveL 4242 to (226.72, 35.59, 69.25) mm, rotated rx 180 ry 0 rz 180 deg; joints [-18.045, 9.924, 62.121, 46.582, 25.243, -43.708]
  MoveL 4243 to (226.72, 35.59, 69.25) mm, rotated rx 180 ry 0 rz 180 deg; joints [-18.045, 9.924, 62.121, 46.582, 25.243, -43.708]
  Call Extruder(198.25916)
  MoveL 4244 to (227.03, 35.63, 69.25) mm, rotated rx -180 ry 0 rz 180 deg; joints [-18.039, 9.978, 62.057, 46.558, 25.246, -43.684]
  MoveL 4245 to (227.03, 35.63, 69.25) mm, rotated rx -180 ry 0 rz 180 deg; joints [-18.039, 9.978, 62.057, 46.558, 25.246, -43.684]
  Call Extruder(198.39309)
  MoveL 4246 to (227.28, 35.68, 69.25) mm, rotated rx -180 ry 0 rz -180 deg; joints [-18.036, 10.023, 62.004, 46.54, 25.249, -43.665]
  MoveL 4247 to (227.28, 35.68, 69.25) mm, rotated rx -180 ry 0 rz -180 deg; joints [-18.036, 10.023, 62.004, 46.54, 25.249, -43.665]
  Call Extruder(198.52763)
  MoveL 4248 to (227.52, 35.73, 69.25) mm, rotated rx -180 ry 0 rz 180 deg; joints [-18.033, 10.068, 61.951, 46.522, 25.252, -43.646]
  MoveL 4249 to (227.52, 35.73, 69.25) mm, rotated rx -180 ry 0 rz 180 deg; joints [-18.033, 10.068, 61.951, 46.522, 25.252, -43.646]
  Call Extruder(198.66277)
  MoveL 4250 to (227.77, 35.78, 69.25) mm, rotated rx 180 ry 0 rz 180 deg; joints [-18.029, 10.113, 61.898, 46.504, 25.255, -43.627]
  MoveL 4251 to (227.77, 35.78, 69.25) mm, rotated rx 180 ry 0 rz 180 deg; joints [-18.029, 10.113, 61.898, 46.504, 25.255, -43.627]
  Call Extruder(198.79853)
  MoveL 4252 to (228.02, 35.83, 69.25) mm, rotated rx 180 ry 0 rz 180 deg; joints [-18.026, 10.158, 61.845, 46.485, 25.258, -43.608]
  MoveL 4253 to (228.02, 35.83, 69.25) mm, rotated rx 180 ry 0 rz 180 deg; joints [-18.026, 10.158, 61.845, 46.485, 25.258, -43.608]
  Call Extruder(198.93490)
  MoveL 4254 to (228.27, 35.88, 69.25) mm, rotated rx 180 ry 0 rz 180 deg; joints [-18.022, 10.203, 61.792, 46.467, 25.262, -43.589]
  MoveL 4255 to (228.27, 35.88, 69.25) mm, rotated rx 180 ry 0 rz 180 deg; joints [-18.022, 10.203, 61.792, 46.467, 25.262, -43.589]
  Call Extruder(199.07188)
  MoveL 4256 to (228.52, 35.93, 69.25) mm, rotated rx 180 ry 0 rz 180 deg; joints [-18.019, 10.248, 61.739, 46.449, 25.265, -43.569]
  MoveL 4257 to (228.52, 35.93, 69.25) mm, rotated rx 180 ry 0 rz 180 deg; joints [-18.019, 10.248, 61.739, 46.449, 25.265, -43.569]
  Call Extruder(199.20947)
  MoveL 4258 to (228.77, 35.98, 69.25) mm, rotated rx 180 ry 0 rz 180 deg; joints [-18.015, 10.293, 61.686, 46.43, 25.268, -43.55]
  MoveL 4259 to (228.77, 35.98, 69.25) mm, rotated rx 180 ry 0 rz 180 deg; joints [-18.015, 10.293, 61.686, 46.43, 25.268, -43.55]
  Call Extruder(199.32318)
  MoveL 4260 to (228.97, 36.03, 69.25) mm, rotated rx 180 ry 0 rz 180 deg; joints [-18.013, 10.33, 61.642, 46.416, 25.271, -43.535]
  MoveL 4261 to (228.97, 36.03, 69.25) mm, rotated rx 180 ry 0 rz 180 deg; joints [-18.013, 10.33, 61.642, 46.416, 25.271, -43.535]
  Call Extruder(199.43735)
  MoveL 4262 to (229.18, 36.07, 69.25) mm, rotated rx 180 ry 0 rz 180 deg; joints [-18.01, 10.367, 61.598, 46.401, 25.274, -43.52]
  MoveL 4263 to (229.18, 36.07, 69.25) mm, rotated rx 180 ry 0 rz 180 deg; joints [-18.01, 10.367, 61.598, 46.401, 25.274, -43.52]
  Call Extruder(199.55198)
  MoveL 4264 to (229.38, 36.12, 69.25) mm, rotated rx 180 ry 0 rz 180 deg; joints [-18.008, 10.404, 61.554, 46.387, 25.277, -43.505]
  MoveL 4265 to (229.38, 36.12, 69.25) mm, rotated rx 180 ry 0 rz 180 deg; joints [-18.008, 10.404, 61.554, 46.387, 25.277, -43.505]
  Call Extruder(199.66705)
  MoveL 4266 to (229.59, 36.16, 69.25) mm, rotated rx 180 ry 0 rz 180 deg; joints [-18.006, 10.442, 61.51, 46.372, 25.28, -43.489]
  MoveL 4267 to (229.59, 36.16, 69.25) mm, rotated rx 180 ry 0 rz 180 deg; joints [-18.006, 10.442, 61.51, 46.372, 25.28, -43.489]
  Call Extruder(199.78928)
  MoveL 4268 to (229.8, 36.22, 69.25) mm, rotated rx 180 ry 0 rz 180 deg; joints [-18.004, 10.481, 61.463, 46.358, 25.284, -43.474]
  MoveL 4269 to (229.8, 36.22, 69.25) mm, rotated rx 180 ry 0 rz 180 deg; joints [-18.004, 10.481, 61.463, 46.358, 25.284, -43.474]
  Call Extruder(199.91895)
  MoveL 4270 to (230.02, 36.28, 69.25) mm, rotated rx 180 ry 0 rz -180 deg; joints [-18.004, 10.523, 61.413, 46.345, 25.289, -43.46]
  MoveL 4271 to (230.02, 36.28, 69.25) mm, rotated rx 180 ry 0 rz -180 deg; joints [-18.004, 10.523, 61.413, 46.345, 25.289, -43.46]
  Call Extruder(200.04918)
  MoveL 4272 to (230.25, 36.35, 69.25) mm, rotated rx -180 ry 0 rz 180 deg; joints [-18.003, 10.565, 61.363, 46.333, 25.294, -43.446]
  MoveL 4273 to (230.25, 36.35, 69.25) mm, rotated rx -180 ry 0 rz 180 deg; joints [-18.003, 10.565, 61.363, 46.333, 25.294, -43.446]
  Call Extruder(200.17998)
  MoveL 4274 to (230.47, 36.42, 69.25) mm, rotated rx -180 ry 0 rz -180 deg; joints [-18.003, 10.607, 61.313, 46.319, 25.299, -43.432]
  MoveL 4275 to (230.47, 36.42, 69.25) mm, rotated rx -180 ry 0 rz -180 deg; joints [-18.003, 10.607, 61.313, 46.319, 25.299, -43.432]
  Call Extruder(200.31134)
  MoveL 4276 to (230.69, 36.49, 69.25) mm, rotated rx -180 ry 0 rz 180 deg; joints [-18.002, 10.649, 61.264, 46.306, 25.305, -43.418]
  MoveL 4277 to (230.69, 36.49, 69.25) mm, rotated rx -180 ry 0 rz 180 deg; joints [-18.002, 10.649, 61.264, 46.306, 25.305, -43.418]
  Call Extruder(200.42676)
  MoveL 4278 to (230.89, 36.55, 69.25) mm, rotated rx -180 ry 0 rz -180 deg; joints [-18.002, 10.686, 61.22, 46.296, 25.309, -43.406]
  MoveL 4279 to (230.89, 36.55, 69.25) mm, rotated rx -180 ry 0 rz -180 deg; joints [-18.002, 10.686, 61.22, 46.296, 25.309, -43.406]
  Call Extruder(200.54265)
  MoveL 4280 to (231.08, 36.61, 69.25) mm, rotated rx -180 ry 0 rz -180 deg; joints [-18.002, 10.722, 61.176, 46.285, 25.314, -43.394]
  MoveL 4281 to (231.08, 36.61, 69.25) mm, rotated rx -180 ry 0 rz -180 deg; joints [-18.002, 10.722, 61.176, 46.285, 25.314, -43.394]
  Call Extruder(200.65547)
  MoveL 4282 to (231.27, 36.68, 69.25) mm, rotated rx 180 ry 0 rz 180 deg; joints [-18.002, 10.758, 61.134, 46.275, 25.319, -43.383]
  MoveL 4283 to (231.27, 36.68, 69.25) mm, rotated rx 180 ry 0 rz 180 deg; joints [-18.002, 10.758, 61.134, 46.275, 25.319, -43.383]
  Call Extruder(200.76517)
  MoveL 4284 to (231.46, 36.73, 69.25) mm, rotated rx 180 ry 0 rz 180 deg; joints [-18.002, 10.793, 61.092, 46.265, 25.323, -43.372]
  MoveL 4285 to (231.46, 36.73, 69.25) mm, rotated rx 180 ry 0 rz 180 deg; joints [-18.002, 10.793, 61.092, 46.265, 25.323, -43.372]
  Call Extruder(200.87528)
  MoveL 4286 to (231.64, 36.79, 69.25) mm, rotated rx -180 ry 0 rz 180 deg; joints [-18.002, 10.827, 61.051, 46.255, 25.328, -43.36]
  MoveL 4287 to (231.64, 36.79, 69.25) mm, rotated rx -180 ry 0 rz 180 deg; joints [-18.002, 10.827, 61.051, 46.255, 25.328, -43.36]
  Call Extruder(201.05724)
  MoveL 4288 to (231.93, 36.91, 69.25) mm, rotated rx 180 ry 0 rz 180 deg; joints [-18.005, 10.884, 60.984, 46.243, 25.338, -43.346]
  MoveL 4289 to (231.93, 36.91, 69.25) mm, rotated rx 180 ry 0 rz 180 deg; joints [-18.005, 10.884, 60.984, 46.243, 25.338, -43.346]
  Call Extruder(201.23996)
  MoveL 4290 to (232.22, 37.03, 69.25) mm, rotated rx -180 ry 0 rz 180 deg; joints [-18.008, 10.941, 60.916, 46.231, 25.347, -43.332]
  MoveL 4291 to (232.22, 37.03, 69.25) mm, rotated rx -180 ry 0 rz 180 deg; joints [-18.008, 10.941, 60.916, 46.231, 25.347, -43.332]
  Call Extruder(201.41037)
  MoveL 4292 to (232.49, 37.15, 69.25) mm, rotated rx -180 ry 0 rz -180 deg; joints [-18.011, 10.994, 60.853, 46.22, 25.356, -43.319]
  MoveL 4293 to (232.49, 37.15, 69.25) mm, rotated rx -180 ry 0 rz -180 deg; joints [-18.011, 10.994, 60.853, 46.22, 25.356, -43.319]
  Call Extruder(201.56837)
  MoveL 4294 to (232.74, 37.26, 69.25) mm, rotated rx -180 ry 0 rz 180 deg; joints [-18.013, 11.043, 60.794, 46.21, 25.365, -43.307]
  MoveL 4295 to (232.74, 37.26, 69.25) mm, rotated rx -180 ry 0 rz 180 deg; joints [-18.013, 11.043, 60.794, 46.21, 25.365, -43.307]
  Call Extruder(201.72697)
  MoveL 4296 to (232.99, 37.36, 69.25) mm, rotated rx -180 ry 0 rz -180 deg; joints [-18.016, 11.092, 60.736, 46.2, 25.373, -43.296]
  MoveL 4297 to (232.99, 37.36, 69.25) mm, rotated rx -180 ry 0 rz -180 deg; joints [-18.016, 11.092, 60.736, 46.2, 25.373, -43.296]
  Call Extruder(201.93314)
  MoveL 4298 to (233.29, 37.54, 69.25) mm, rotated rx -180 ry 0 rz 180 deg; joints [-18.024, 11.154, 60.661, 46.196, 25.387, -43.288]
  MoveL 4299 to (233.29, 37.54, 69.25) mm, rotated rx -180 ry 0 rz 180 deg; joints [-18.024, 11.154, 60.661, 46.196, 25.387, -43.288]
  Call Extruder(202.14008)
  MoveL 4300 to (233.6, 37.71, 69.25) mm, rotated rx 180 ry 0 rz 180 deg; joints [-18.033, 11.216, 60.587, 46.191, 25.402, -43.28]
  MoveL 4301 to (233.6, 37.71, 69.25) mm, rotated rx 180 ry 0 rz 180 deg; joints [-18.033, 11.216, 60.587, 46.191, 25.402, -43.28]
  Call Extruder(202.34781)
  MoveL 4302 to (233.9, 37.89, 69.25) mm, rotated rx -180 ry 0 rz -180 deg; joints [-18.041, 11.278, 60.512, 46.186, 25.416, -43.271]
  MoveL 4303 to (233.9, 37.89, 69.25) mm, rotated rx -180 ry 0 rz -180 deg; joints [-18.041, 11.278, 60.512, 46.186, 25.416, -43.271]
  Call Extruder(202.55631)
  MoveL 4304 to (234.21, 38.06, 69.25) mm, rotated rx 180 ry 0 rz 180 deg; joints [-18.049, 11.341, 60.437, 46.181, 25.43, -43.263]
  MoveL 4305 to (234.21, 38.06, 69.25) mm, rotated rx 180 ry 0 rz 180 deg; joints [-18.049, 11.341, 60.437, 46.181, 25.43, -43.263]
  Call Extruder(202.73585)
  MoveL 4306 to (234.45, 38.24, 69.25) mm, rotated rx 180 ry 0 rz 180 deg; joints [-18.06, 11.393, 60.374, 46.183, 25.445, -43.261]
  MoveL 4307 to (234.45, 38.24, 69.25) mm, rotated rx 180 ry 0 rz 180 deg; joints [-18.06, 11.393, 60.374, 46.183, 25.445, -43.261]
  Call Extruder(203.06927)
  MoveL 4308 to (234.9, 38.57, 69.25) mm, rotated rx -180 ry 0 rz -180 deg; joints [-18.079, 11.49, 60.258, 46.186, 25.472, -43.258]
  MoveL 4309 to (234.9, 38.57, 69.25) mm, rotated rx -180 ry 0 rz -180 deg; joints [-18.079, 11.49, 60.258, 46.186, 25.472, -43.258]
  Call Extruder(203.40387)
  MoveL 4310 to (235.35, 38.9, 69.25) mm, rotated rx 180 ry 0 rz -180 deg; joints [-18.099, 11.587, 60.141, 46.189, 25.499, -43.255]
  Call Extruder(204.23182)
  MoveL 4311 to (236.39, 39.81, 69.25) mm, rotated rx 180 ry 0 rz -180 deg; joints [-18.16, 11.819, 59.861, 46.22, 25.575, -43.268]
  Call Extruder(205.05976)
  MoveL 4312 to (237.3, 40.85, 69.25) mm, rotated rx -180 ry 0 rz -180 deg; joints [-18.24, 12.037, 59.596, 46.284, 25.661, -43.311]
  Call Extruder(205.22706)
  MoveL 4313 to (237.47, 41.07, 69.25) mm, rotated rx 180 ry 0 rz 180 deg; joints [-18.258, 12.079, 59.545, 46.302, 25.68, -43.324]
  MoveL 4314 to (237.47, 41.07, 69.25) mm, rotated rx 180 ry 0 rz 180 deg; joints [-18.258, 12.079, 59.545, 46.302, 25.68, -43.324]
  Call Extruder(205.56048)
  MoveL 4315 to (237.79, 41.52, 69.25) mm, rotated rx -180 ry 0 rz 180 deg; joints [-18.295, 12.162, 59.444, 46.336, 25.717, -43.349]
  MoveL 4316 to (237.79, 41.52, 69.25) mm, rotated rx -180 ry 0 rz 180 deg; joints [-18.295, 12.162, 59.444, 46.336, 25.717, -43.349]
  Call Extruder(205.89270)
  MoveL 4317 to (238.12, 41.97, 69.25) mm, rotated rx -180 ry 0 rz 180 deg; joints [-18.332, 12.246, 59.342, 46.37, 25.755, -43.374]
  MoveL 4318 to (238.12, 41.97, 69.25) mm, rotated rx -180 ry 0 rz 180 deg; joints [-18.332, 12.246, 59.342, 46.37, 25.755, -43.374]
  Call Extruder(206.01040)
  MoveL 4319 to (238.22, 42.15, 69.25) mm, rotated rx 180 ry 0 rz 180 deg; joints [-18.346, 12.274, 59.308, 46.386, 25.769, -43.387]
  MoveL 4320 to (238.22, 42.15, 69.25) mm, rotated rx 180 ry 0 rz 180 deg; joints [-18.346, 12.274, 59.308, 46.386, 25.769, -43.387]
  Call Extruder(206.21813)
  MoveL 4321 to (238.4, 42.45, 69.25) mm, rotated rx 180 ry 0 rz 180 deg; joints [-18.373, 12.322, 59.249, 46.414, 25.795, -43.409]
  MoveL 4322 to (238.4, 42.45, 69.25) mm, rotated rx 180 ry 0 rz 180 deg; joints [-18.373, 12.322, 59.249, 46.414, 25.795, -43.409]
  Call Extruder(206.42507)
  MoveL 4323 to (238.57, 42.75, 69.25) mm, rotated rx 180 ry 0 rz 180 deg; joints [-18.399, 12.371, 59.19, 46.442, 25.82, -43.43]
  MoveL 4324 to (238.57, 42.75, 69.25) mm, rotated rx 180 ry 0 rz 180 deg; joints [-18.399, 12.371, 59.19, 46.442, 25.82, -43.43]
  Call Extruder(206.63124)
  MoveL 4325 to (238.75, 43.06, 69.25) mm, rotated rx -180 ry 0 rz 180 deg; joints [-18.425, 12.419, 59.131, 46.47, 25.846, -43.452]
  MoveL 4326 to (238.75, 43.06, 69.25) mm, rotated rx -180 ry 0 rz 180 deg; joints [-18.425, 12.419, 59.131, 46.47, 25.846, -43.452]
  Call Extruder(206.81293)
  MoveL 4327 to (238.89, 43.34, 69.25) mm, rotated rx 180 ry 0 rz 180 deg; joints [-18.45, 12.46, 59.081, 46.497, 25.869, -43.473]
  MoveL 4328 to (238.89, 43.34, 69.25) mm, rotated rx 180 ry 0 rz 180 deg; joints [-18.45, 12.46, 59.081, 46.497, 25.869, -43.473]
  Call Extruder(206.97094)
  MoveL 4329 to (239, 43.58, 69.25) mm, rotated rx -180 ry 0 rz 180 deg; joints [-18.472, 12.494, 59.04, 46.524, 25.889, -43.495]
  MoveL 4330 to (239, 43.58, 69.25) mm, rotated rx -180 ry 0 rz 180 deg; joints [-18.472, 12.494, 59.04, 46.524, 25.889, -43.495]
  Call Extruder(207.12835)
  MoveL 4331 to (239.11, 43.83, 69.25) mm, rotated rx 180 ry 0 rz -180 deg; joints [-18.495, 12.527, 58.999, 46.55, 25.91, -43.517]
  MoveL 4332 to (239.11, 43.83, 69.25) mm, rotated rx 180 ry 0 rz -180 deg; joints [-18.495, 12.527, 58.999, 46.55, 25.91, -43.517]
  Call Extruder(207.31106)
  MoveL 4333 to (239.23, 44.12, 69.25) mm, rotated rx -180 ry 0 rz 180 deg; joints [-18.522, 12.566, 58.952, 46.582, 25.935, -43.543]
  MoveL 4334 to (239.23, 44.12, 69.25) mm, rotated rx -180 ry 0 rz 180 deg; joints [-18.522, 12.566, 58.952, 46.582, 25.935, -43.543]
  Call Extruder(207.49302)
  MoveL 4335 to (239.35, 44.42, 69.25) mm, rotated rx 180 ry 0 rz 180 deg; joints [-18.549, 12.604, 58.905, 46.613, 25.959, -43.568]
  MoveL 4336 to (239.35, 44.42, 69.25) mm, rotated rx 180 ry 0 rz 180 deg; joints [-18.549, 12.604, 58.905, 46.613, 25.959, -43.568]
  Call Extruder(207.64035)
  MoveL 4337 to (239.44, 44.66, 69.25) mm, rotated rx -180 ry 0 rz -180 deg; joints [-18.571, 12.634, 58.868, 46.64, 25.979, -43.59]
  MoveL 4338 to (239.44, 44.66, 69.25) mm, rotated rx -180 ry 0 rz -180 deg; joints [-18.571, 12.634, 58.868, 46.64, 25.979, -43.59]
  Call Extruder(207.75359)
  MoveL 4339 to (239.5, 44.85, 69.25) mm, rotated rx -180 ry 0 rz 180 deg; joints [-18.589, 12.657, 58.841, 46.662, 25.995, -43.608]
  MoveL 4340 to (239.5, 44.85, 69.25) mm, rotated rx -180 ry 0 rz 180 deg; joints [-18.589, 12.657, 58.841, 46.662, 25.995, -43.608]
  Call Extruder(207.86638)
  MoveL 4341 to (239.56, 45.03, 69.25) mm, rotated rx -180 ry 0 rz 180 deg; joints [-18.607, 12.678, 58.814, 46.684, 26.01, -43.627]
  MoveL 4342 to (239.56, 45.03, 69.25) mm, rotated rx -180 ry 0 rz 180 deg; joints [-18.607, 12.678, 58.814, 46.684, 26.01, -43.627]
  Call Extruder(207.97872)
  MoveL 4343 to (239.62, 45.22, 69.25) mm, rotated rx -180 ry 0 rz 180 deg; joints [-18.625, 12.7, 58.787, 46.707, 26.026, -43.645]
  MoveL 4344 to (239.62, 45.22, 69.25) mm, rotated rx -180 ry 0 rz 180 deg; joints [-18.625, 12.7, 58.787, 46.707, 26.026, -43.645]
  Call Extruder(208.09063)
  MoveL 4345 to (239.68, 45.41, 69.25) mm, rotated rx -180 ry 0 rz 180 deg; joints [-18.642, 12.722, 58.76, 46.729, 26.042, -43.663]
  MoveL 4346 to (239.68, 45.41, 69.25) mm, rotated rx -180 ry 0 rz 180 deg; joints [-18.642, 12.722, 58.76, 46.729, 26.042, -43.663]
  Call Extruder(208.21203)
  MoveL 4347 to (239.75, 45.62, 69.25) mm, rotated rx 180 ry 0 rz -180 deg; joints [-18.662, 12.746, 58.731, 46.753, 26.059, -43.683]
  MoveL 4348 to (239.75, 45.62, 69.25) mm, rotated rx 180 ry 0 rz -180 deg; joints [-18.662, 12.746, 58.731, 46.753, 26.059, -43.683]
  Call Extruder(208.34282)
  MoveL 4349 to (239.82, 45.84, 69.25) mm, rotated rx -180 ry 0 rz 180 deg; joints [-18.683, 12.771, 58.7, 46.779, 26.078, -43.705]
  MoveL 4350 to (239.82, 45.84, 69.25) mm, rotated rx -180 ry 0 rz 180 deg; joints [-18.683, 12.771, 58.7, 46.779, 26.078, -43.705]
  Call Extruder(208.47304)
  MoveL 4351 to (239.88, 46.06, 69.25) mm, rotated rx 180 ry 0 rz 180 deg; joints [-18.705, 12.797, 58.669, 46.806, 26.096, -43.727]
  MoveL 4352 to (239.88, 46.06, 69.25) mm, rotated rx 180 ry 0 rz 180 deg; joints [-18.705, 12.797, 58.669, 46.806, 26.096, -43.727]
  Call Extruder(208.60270)
  MoveL 4353 to (239.95, 46.29, 69.25) mm, rotated rx -180 ry 0 rz 180 deg; joints [-18.726, 12.822, 58.638, 46.832, 26.115, -43.749]
  MoveL 4354 to (239.95, 46.29, 69.25) mm, rotated rx -180 ry 0 rz 180 deg; joints [-18.726, 12.822, 58.638, 46.832, 26.115, -43.749]
  Call Extruder(208.73180)
  MoveL 4355 to (240.02, 46.51, 69.25) mm, rotated rx 180 ry 0 rz 180 deg; joints [-18.747, 12.847, 58.607, 46.859, 26.134, -43.771]
  MoveL 4356 to (240.02, 46.51, 69.25) mm, rotated rx 180 ry 0 rz 180 deg; joints [-18.747, 12.847, 58.607, 46.859, 26.134, -43.771]
  Call Extruder(208.84685)
  MoveL 4357 to (240.06, 46.72, 69.25) mm, rotated rx 180 ry 0 rz 180 deg; joints [-18.767, 12.868, 58.582, 46.885, 26.151, -43.793]
  MoveL 4358 to (240.06, 46.72, 69.25) mm, rotated rx 180 ry 0 rz 180 deg; joints [-18.767, 12.868, 58.582, 46.885, 26.151, -43.793]
  Call Extruder(208.96145)
  MoveL 4359 to (240.11, 46.92, 69.25) mm, rotated rx 180 ry 0 rz 180 deg; joints [-18.787, 12.888, 58.557, 46.91, 26.168, -43.814]
  MoveL 4360 to (240.11, 46.92, 69.25) mm, rotated rx 180 ry 0 rz 180 deg; joints [-18.787, 12.888, 58.557, 46.91, 26.168, -43.814]
  Call Extruder(209.07560)
  MoveL 4361 to (240.15, 47.12, 69.25) mm, rotated rx -180 ry 0 rz 180 deg; joints [-18.807, 12.908, 58.532, 46.936, 26.185, -43.836]
  MoveL 4362 to (240.15, 47.12, 69.25) mm, rotated rx -180 ry 0 rz 180 deg; joints [-18.807, 12.908, 58.532, 46.936, 26.185, -43.836]
  Call Extruder(209.18930)
  MoveL 4363 to (240.2, 47.33, 69.25) mm, rotated rx -180 ry 0 rz 180 deg; joints [-18.827, 12.928, 58.507, 46.962, 26.202, -43.858]
  MoveL 4364 to (240.2, 47.33, 69.25) mm, rotated rx -180 ry 0 rz 180 deg; joints [-18.827, 12.928, 58.507, 46.962, 26.202, -43.858]
  Call Extruder(209.31471)
  MoveL 4365 to (240.24, 47.56, 69.25) mm, rotated rx -180 ry 0 rz -180 deg; joints [-18.85, 12.95, 58.48, 46.991, 26.221, -43.882]
  MoveL 4366 to (240.24, 47.56, 69.25) mm, rotated rx -180 ry 0 rz -180 deg; joints [-18.85, 12.95, 58.48, 46.991, 26.221, -43.882]
  Call Extruder(209.45169)
  MoveL 4367 to (240.29, 47.8, 69.25) mm, rotated rx -180 ry 0 rz 180 deg; joints [-18.874, 12.974, 58.451, 47.023, 26.242, -43.909]
  MoveL 4368 to (240.29, 47.8, 69.25) mm, rotated rx -180 ry 0 rz 180 deg; joints [-18.874, 12.974, 58.451, 47.023, 26.242, -43.909]
  Call Extruder(209.58805)
  MoveL 4369 to (240.34, 48.05, 69.25) mm, rotated rx 180 ry 0 rz 180 deg; joints [-18.899, 12.998, 58.422, 47.055, 26.262, -43.936]
  MoveL 4370 to (240.34, 48.05, 69.25) mm, rotated rx 180 ry 0 rz 180 deg; joints [-18.899, 12.998, 58.422, 47.055, 26.262, -43.936]
  Call Extruder(209.72381)
  MoveL 4371 to (240.39, 48.3, 69.25) mm, rotated rx 180 ry 0 rz 180 deg; joints [-18.923, 13.022, 58.392, 47.087, 26.283, -43.962]
  MoveL 4372 to (240.39, 48.3, 69.25) mm, rotated rx 180 ry 0 rz 180 deg; joints [-18.923, 13.022, 58.392, 47.087, 26.283, -43.962]
  Call Extruder(209.85896)
  MoveL 4373 to (240.44, 48.55, 69.25) mm, rotated rx 180 ry 0 rz 180 deg; joints [-18.948, 13.046, 58.363, 47.118, 26.304, -43.989]
  MoveL 4374 to (240.44, 48.55, 69.25) mm, rotated rx 180 ry 0 rz 180 deg; joints [-18.948, 13.046, 58.363, 47.118, 26.304, -43.989]
  Call Extruder(209.99349)
  MoveL 4375 to (240.49, 48.8, 69.25) mm, rotated rx 180 ry 0 rz -180 deg; joints [-18.973, 13.07, 58.333, 47.15, 26.325, -44.015]
  MoveL 4376 to (240.49, 48.8, 69.25) mm, rotated rx 180 ry 0 rz -180 deg; joints [-18.973, 13.07, 58.333, 47.15, 26.325, -44.015]
  Call Extruder(210.12742)
  MoveL 4377 to (240.54, 49.05, 69.25) mm, rotated rx -180 ry 0 rz 180 deg; joints [-18.997, 13.093, 58.304, 47.181, 26.346, -44.042]
  MoveL 4378 to (240.54, 49.05, 69.25) mm, rotated rx -180 ry 0 rz 180 deg; joints [-18.997, 13.093, 58.304, 47.181, 26.346, -44.042]
  Call Extruder(210.27529)
  MoveL 4379 to (240.59, 49.33, 69.25) mm, rotated rx 180 ry 0 rz 180 deg; joints [-19.025, 13.119, 58.272, 47.217, 26.369, -44.072]
  MoveL 4380 to (240.59, 49.33, 69.25) mm, rotated rx 180 ry 0 rz 180 deg; joints [-19.025, 13.119, 58.272, 47.217, 26.369, -44.072]
  Call Extruder(210.43703)
  MoveL 4381 to (240.64, 49.63, 69.25) mm, rotated rx 180 ry 0 rz 180 deg; joints [-19.055, 13.147, 58.238, 47.257, 26.394, -44.106]
  MoveL 4382 to (240.64, 49.63, 69.25) mm, rotated rx 180 ry 0 rz 180 deg; joints [-19.055, 13.147, 58.238, 47.257, 26.394, -44.106]
  Call Extruder(210.59805)
  MoveL 4383 to (240.69, 49.94, 69.25) mm, rotated rx 180 ry 0 rz 180 deg; joints [-19.086, 13.174, 58.205, 47.297, 26.42, -44.139]
  MoveL 4384 to (240.69, 49.94, 69.25) mm, rotated rx 180 ry 0 rz 180 deg; joints [-19.086, 13.174, 58.205, 47.297, 26.42, -44.139]
  Call Extruder(210.75834)
  MoveL 4385 to (240.74, 50.24, 69.25) mm, rotated rx -180 ry 0 rz 180 deg; joints [-19.116, 13.201, 58.171, 47.336, 26.445, -44.172]
  MoveL 4386 to (240.74, 50.24, 69.25) mm, rotated rx -180 ry 0 rz 180 deg; joints [-19.116, 13.201, 58.171, 47.336, 26.445, -44.172]
  Call Extruder(210.91790)
  MoveL 4387 to (240.78, 50.55, 69.25) mm, rotated rx -180 ry 0 rz 180 deg; joints [-19.146, 13.229, 58.137, 47.376, 26.471, -44.206]
  MoveL 4388 to (240.78, 50.55, 69.25) mm, rotated rx -180 ry 0 rz 180 deg; joints [-19.146, 13.229, 58.137, 47.376, 26.471, -44.206]
  Call Extruder(211.07673)
  MoveL 4389 to (240.83, 50.86, 69.25) mm, rotated rx 180 ry 0 rz 180 deg; joints [-19.177, 13.256, 58.103, 47.415, 26.497, -44.239]
  MoveL 4390 to (240.83, 50.86, 69.25) mm, rotated rx 180 ry 0 rz 180 deg; joints [-19.177, 13.256, 58.103, 47.415, 26.497, -44.239]
  Call Extruder(211.25540)
  MoveL 4391 to (240.88, 51.2, 69.25) mm, rotated rx -180 ry 0 rz 180 deg; joints [-19.212, 13.286, 58.066, 47.46, 26.526, -44.277]
  MoveL 4392 to (240.88, 51.2, 69.25) mm, rotated rx -180 ry 0 rz 180 deg; joints [-19.212, 13.286, 58.066, 47.46, 26.526, -44.277]
  Call Extruder(211.45384)
  MoveL 4393 to (240.92, 51.59, 69.25) mm, rotated rx 180 ry 0 rz 180 deg; joints [-19.251, 13.318, 58.026, 47.512, 26.558, -44.321]
  MoveL 4394 to (240.92, 51.59, 69.25) mm, rotated rx 180 ry 0 rz 180 deg; joints [-19.251, 13.318, 58.026, 47.512, 26.558, -44.321]
  Call Extruder(211.65142)
  MoveL 4395 to (240.97, 51.98, 69.25) mm, rotated rx 180 ry 0 rz 180 deg; joints [-19.29, 13.35, 57.986, 47.563, 26.591, -44.364]
  MoveL 4396 to (240.97, 51.98, 69.25) mm, rotated rx 180 ry 0 rz 180 deg; joints [-19.29, 13.35, 57.986, 47.563, 26.591, -44.364]
  Call Extruder(211.84813)
  MoveL 4397 to (241.02, 52.36, 69.25) mm, rotated rx -180 ry 0 rz -180 deg; joints [-19.329, 13.383, 57.946, 47.614, 26.623, -44.407]
  MoveL 4398 to (241.02, 52.36, 69.25) mm, rotated rx -180 ry 0 rz -180 deg; joints [-19.329, 13.383, 57.946, 47.614, 26.623, -44.407]
  Call Extruder(212.04396)
  MoveL 4399 to (241.06, 52.75, 69.25) mm, rotated rx 180 ry 0 rz 180 deg; joints [-19.368, 13.415, 57.906, 47.665, 26.656, -44.45]
  MoveL 4400 to (241.06, 52.75, 69.25) mm, rotated rx 180 ry 0 rz 180 deg; joints [-19.368, 13.415, 57.906, 47.665, 26.656, -44.45]
  Call Extruder(212.33940)
  MoveL 4401 to (241.11, 53.34, 69.25) mm, rotated rx -180 ry 0 rz 180 deg; joints [-19.428, 13.46, 57.85, 47.745, 26.705, -44.517]
  MoveL 4402 to (241.11, 53.34, 69.25) mm, rotated rx -180 ry 0 rz 180 deg; joints [-19.428, 13.46, 57.85, 47.745, 26.705, -44.517]
  Call Extruder(212.63351)
  MoveL 4403 to (241.16, 53.93, 69.25) mm, rotated rx -180 ry 0 rz 180 deg; joints [-19.488, 13.506, 57.794, 47.824, 26.755, -44.584]
  MoveL 4404 to (241.16, 53.93, 69.25) mm, rotated rx -180 ry 0 rz 180 deg; joints [-19.488, 13.506, 57.794, 47.824, 26.755, -44.584]
  Call Extruder(212.92629)
  MoveL 4405 to (241.2, 54.52, 69.25) mm, rotated rx -180 ry 0 rz 180 deg; joints [-19.548, 13.551, 57.737, 47.903, 26.804, -44.651]
  MoveL 4406 to (241.2, 54.52, 69.25) mm, rotated rx -180 ry 0 rz 180 deg; joints [-19.548, 13.551, 57.737, 47.903, 26.804, -44.651]
  Call Extruder(213.49974)
  MoveL 4407 to (241.25, 55.68, 69.25) mm, rotated rx -180 ry 0 rz 180 deg; joints [-19.668, 13.633, 57.636, 48.062, 26.902, -44.787]
  MoveL 4408 to (241.25, 55.68, 69.25) mm, rotated rx -180 ry 0 rz 180 deg; joints [-19.668, 13.633, 57.636, 48.062, 26.902, -44.787]
  Call Extruder(214.21357)
  MoveL 4409 to (241.29, 57.14, 69.25) mm, rotated rx 180 ry 0 rz 180 deg; joints [-19.819, 13.733, 57.511, 48.262, 27.024, -44.957]
  Call Extruder(256.27845)
  MoveL 4410 to (241.29, 142.86, 69.25) mm, rotated rx -180 ry 0 rz -180 deg; joints [-28.232, 20.913, 48.106, 56.301, 34.652, -50.968]
  Call Extruder(256.70688)
  MoveL 4411 to (241.27, 143.73, 69.25) mm, rotated rx 180 ry 0 rz 180 deg; joints [-28.313, 21.002, 47.982, 56.349, 34.733, -50.992]
  MoveL 4412 to (241.27, 143.73, 69.25) mm, rotated rx 180 ry 0 rz 180 deg; joints [-28.313, 21.002, 47.982, 56.349, 34.733, -50.992]
  Call Extruder(257.28033)
  MoveL 4413 to (241.23, 144.9, 69.25) mm, rotated rx -180 ry 0 rz -180 deg; joints [-28.421, 21.118, 47.822, 56.416, 34.842, -51.026]
  MoveL 4414 to (241.23, 144.9, 69.25) mm, rotated rx -180 ry 0 rz -180 deg; joints [-28.421, 21.118, 47.822, 56.416, 34.842, -51.026]
  Call Extruder(257.71467)
  MoveL 4415 to (241.18, 145.77, 69.25) mm, rotated rx -180 ry 0 rz 180 deg; joints [-28.503, 21.204, 47.704, 56.468, 34.924, -51.053]
  MoveL 4416 to (241.18, 145.77, 69.25) mm, rotated rx -180 ry 0 rz 180 deg; joints [-28.503, 21.204, 47.704, 56.468, 34.924, -51.053]
  Call Extruder(258.00878)
  MoveL 4417 to (241.13, 146.36, 69.25) mm, rotated rx 180 ry 0 rz -180 deg; joints [-28.559, 21.258, 47.629, 56.504, 34.979, -51.073]
  MoveL 4418 to (241.13, 146.36, 69.25) mm, rotated rx 180 ry 0 rz -180 deg; joints [-28.559, 21.258, 47.629, 56.504, 34.979, -51.073]
  Call Extruder(258.30422)
  MoveL 4419 to (241.09, 146.95, 69.25) mm, rotated rx 180 ry 0 rz 180 deg; joints [-28.615, 21.313, 47.553, 56.54, 35.034, -51.092]
  MoveL 4420 to (241.09, 146.95, 69.25) mm, rotated rx 180 ry 0 rz 180 deg; joints [-28.615, 21.313, 47.553, 56.54, 35.034, -51.092]
  Call Extruder(258.55047)
  MoveL 4421 to (241.04, 147.44, 69.25) mm, rotated rx 180 ry 0 rz 180 deg; joints [-28.662, 21.357, 47.492, 56.571, 35.08, -51.11]
  MoveL 4422 to (241.04, 147.44, 69.25) mm, rotated rx 180 ry 0 rz 180 deg; joints [-28.662, 21.357, 47.492, 56.571, 35.08, -51.11]
  Call Extruder(258.74718)
  MoveL 4423 to (240.99, 147.83, 69.25) mm, rotated rx 180 ry 0 rz 180 deg; joints [-28.7, 21.391, 47.446, 56.597, 35.116, -51.125]
  MoveL 4424 to (240.99, 147.83, 69.25) mm, rotated rx 180 ry 0 rz 180 deg; joints [-28.7, 21.391, 47.446, 56.597, 35.116, -51.125]
  Call Extruder(258.94475)
  MoveL 4425 to (240.95, 148.22, 69.25) mm, rotated rx 180 ry 0 rz -180 deg; joints [-28.737, 21.424, 47.4, 56.623, 35.152, -51.139]
  MoveL 4426 to (240.95, 148.22, 69.25) mm, rotated rx 180 ry 0 rz -180 deg; joints [-28.737, 21.424, 47.4, 56.623, 35.152, -51.139]
  Call Extruder(259.14319)
  MoveL 4427 to (240.9, 148.6, 69.25) mm, rotated rx -180 ry 0 rz -180 deg; joints [-28.774, 21.457, 47.353, 56.648, 35.189, -51.154]
  MoveL 4428 to (240.9, 148.6, 69.25) mm, rotated rx -180 ry 0 rz -180 deg; joints [-28.774, 21.457, 47.353, 56.648, 35.189, -51.154]
  Call Extruder(259.34250)
  MoveL 4429 to (240.86, 148.99, 69.25) mm, rotated rx -180 ry 0 rz 180 deg; joints [-28.812, 21.491, 47.307, 56.673, 35.225, -51.168]
  MoveL 4430 to (240.86, 148.99, 69.25) mm, rotated rx -180 ry 0 rz 180 deg; joints [-28.812, 21.491, 47.307, 56.673, 35.225, -51.168]
  Call Extruder(259.50134)
  MoveL 4431 to (240.81, 149.3, 69.25) mm, rotated rx 180 ry 0 rz 180 deg; joints [-28.842, 21.515, 47.273, 56.695, 35.253, -51.182]
  MoveL 4432 to (240.81, 149.3, 69.25) mm, rotated rx 180 ry 0 rz 180 deg; joints [-28.842, 21.515, 47.273, 56.695, 35.253, -51.182]
  Call Extruder(259.66090)
  MoveL 4433 to (240.76, 149.6, 69.25) mm, rotated rx 180 ry 0 rz 180 deg; joints [-28.872, 21.539, 47.24, 56.717, 35.282, -51.195]
  MoveL 4434 to (240.76, 149.6, 69.25) mm, rotated rx 180 ry 0 rz 180 deg; joints [-28.872, 21.539, 47.24, 56.717, 35.282, -51.195]
  Call Extruder(259.82119)
  MoveL 4435 to (240.71, 149.91, 69.25) mm, rotated rx 180 ry 0 rz 180 deg; joints [-28.902, 21.563, 47.206, 56.738, 35.311, -51.208]
  MoveL 4436 to (240.71, 149.91, 69.25) mm, rotated rx 180 ry 0 rz 180 deg; joints [-28.902, 21.563, 47.206, 56.738, 35.311, -51.208]
  Call Extruder(259.98220)
  MoveL 4437 to (240.66, 150.21, 69.25) mm, rotated rx -180 ry 0 rz 180 deg; joints [-28.932, 21.587, 47.173, 56.76, 35.339, -51.221]
  MoveL 4438 to (240.66, 150.21, 69.25) mm, rotated rx -180 ry 0 rz 180 deg; joints [-28.932, 21.587, 47.173, 56.76, 35.339, -51.221]
  Call Extruder(260.14395)
  MoveL 4439 to (240.61, 150.52, 69.25) mm, rotated rx -180 ry 0 rz 180 deg; joints [-28.962, 21.611, 47.139, 56.781, 35.368, -51.234]
  MoveL 4440 to (240.61, 150.52, 69.25) mm, rotated rx -180 ry 0 rz 180 deg; joints [-28.962, 21.611, 47.139, 56.781, 35.368, -51.234]
  Call Extruder(260.30642)
  MoveL 4441 to (240.56, 150.83, 69.25) mm, rotated rx -180 ry 0 rz -180 deg; joints [-28.993, 21.636, 47.105, 56.803, 35.397, -51.247]
  MoveL 4442 to (240.56, 150.83, 69.25) mm, rotated rx -180 ry 0 rz -180 deg; joints [-28.993, 21.636, 47.105, 56.803, 35.397, -51.247]
  Call Extruder(260.44035)
  MoveL 4443 to (240.52, 151.08, 69.25) mm, rotated rx 180 ry 0 rz 180 deg; joints [-29.017, 21.654, 47.081, 56.821, 35.42, -51.258]
  MoveL 4444 to (240.52, 151.08, 69.25) mm, rotated rx 180 ry 0 rz 180 deg; joints [-29.017, 21.654, 47.081, 56.821, 35.42, -51.258]
  Call Extruder(260.57488)
  MoveL 4445 to (240.47, 151.32, 69.25) mm, rotated rx 180 ry 0 rz 180 deg; joints [-29.043, 21.671, 47.056, 56.84, 35.443, -51.27]
  MoveL 4446 to (240.47, 151.32, 69.25) mm, rotated rx 180 ry 0 rz 180 deg; joints [-29.043, 21.671, 47.056, 56.84, 35.443, -51.27]
  Call Extruder(260.71003)
  MoveL 4447 to (240.42, 151.57, 69.25) mm, rotated rx 180 ry 0 rz -180 deg; joints [-29.067, 21.689, 47.031, 56.859, 35.466, -51.282]
  MoveL 4448 to (240.42, 151.57, 69.25) mm, rotated rx 180 ry 0 rz -180 deg; joints [-29.067, 21.689, 47.031, 56.859, 35.466, -51.282]
  Call Extruder(260.84579)
  MoveL 4449 to (240.37, 151.82, 69.25) mm, rotated rx 180 ry 0 rz 180 deg; joints [-29.092, 21.707, 47.006, 56.878, 35.49, -51.294]
  MoveL 4450 to (240.37, 151.82, 69.25) mm, rotated rx 180 ry 0 rz 180 deg; joints [-29.092, 21.707, 47.006, 56.878, 35.49, -51.294]
  Call Extruder(260.98215)
  MoveL 4451 to (240.32, 152.07, 69.25) mm, rotated rx -180 ry 0 rz 180 deg; joints [-29.117, 21.725, 46.981, 56.896, 35.513, -51.306]
  MoveL 4452 to (240.32, 152.07, 69.25) mm, rotated rx -180 ry 0 rz 180 deg; joints [-29.117, 21.725, 46.981, 56.896, 35.513, -51.306]
  Call Extruder(261.11913)
  MoveL 4453 to (240.27, 152.32, 69.25) mm, rotated rx 180 ry 0 rz -180 deg; joints [-29.142, 21.743, 46.956, 56.915, 35.536, -51.318]
  MoveL 4454 to (240.27, 152.32, 69.25) mm, rotated rx 180 ry 0 rz -180 deg; joints [-29.142, 21.743, 46.956, 56.915, 35.536, -51.318]
  Call Extruder(261.25672)
  MoveL 4455 to (240.22, 152.57, 69.25) mm, rotated rx 180 ry 0 rz -180 deg; joints [-29.167, 21.761, 46.931, 56.933, 35.56, -51.329]
  MoveL 4456 to (240.22, 152.57, 69.25) mm, rotated rx 180 ry 0 rz -180 deg; joints [-29.167, 21.761, 46.931, 56.933, 35.56, -51.329]
  Call Extruder(261.37042)
  MoveL 4457 to (240.17, 152.77, 69.25) mm, rotated rx 180 ry 0 rz 180 deg; joints [-29.188, 21.775, 46.911, 56.949, 35.579, -51.339]
  MoveL 4458 to (240.17, 152.77, 69.25) mm, rotated rx 180 ry 0 rz 180 deg; joints [-29.188, 21.775, 46.911, 56.949, 35.579, -51.339]
  Call Extruder(261.48457)
  MoveL 4459 to (240.13, 152.98, 69.25) mm, rotated rx 180 ry 0 rz 180 deg; joints [-29.209, 21.789, 46.892, 56.965, 35.598, -51.349]
  MoveL 4460 to (240.13, 152.98, 69.25) mm, rotated rx 180 ry 0 rz 180 deg; joints [-29.209, 21.789, 46.892, 56.965, 35.598, -51.349]
  Call Extruder(261.59917)
  MoveL 4461 to (240.08, 153.18, 69.25) mm, rotated rx 180 ry 0 rz 180 deg; joints [-29.229, 21.803, 46.873, 56.981, 35.617, -51.36]
  MoveL 4462 to (240.08, 153.18, 69.25) mm, rotated rx 180 ry 0 rz 180 deg; joints [-29.229, 21.803, 46.873, 56.981, 35.617, -51.36]
  Call Extruder(261.71422)
  MoveL 4463 to (240.04, 153.39, 69.25) mm, rotated rx 180 ry 0 rz 180 deg; joints [-29.25, 21.817, 46.853, 56.996, 35.636, -51.369]
  MoveL 4464 to (240.04, 153.39, 69.25) mm, rotated rx 180 ry 0 rz 180 deg; joints [-29.25, 21.817, 46.853, 56.996, 35.636, -51.369]
  Call Extruder(261.83645)
  MoveL 4465 to (239.98, 153.6, 69.25) mm, rotated rx 180 ry 0 rz 180 deg; joints [-29.272, 21.83, 46.835, 57.014, 35.656, -51.381]
  MoveL 4466 to (239.98, 153.6, 69.25) mm, rotated rx 180 ry 0 rz 180 deg; joints [-29.272, 21.83, 46.835, 57.014, 35.656, -51.381]
  Call Extruder(261.96611)
  MoveL 4467 to (239.92, 153.82, 69.25) mm, rotated rx -180 ry 0 rz -180 deg; joints [-29.296, 21.842, 46.819, 57.034, 35.677, -51.395]
  MoveL 4468 to (239.92, 153.82, 69.25) mm, rotated rx -180 ry 0 rz -180 deg; joints [-29.296, 21.842, 46.819, 57.034, 35.677, -51.395]
  Call Extruder(262.09633)
  MoveL 4469 to (239.85, 154.05, 69.25) mm, rotated rx 180 ry 0 rz -180 deg; joints [-29.319, 21.853, 46.803, 57.054, 35.698, -51.409]
  MoveL 4470 to (239.85, 154.05, 69.25) mm, rotated rx 180 ry 0 rz -180 deg; joints [-29.319, 21.853, 46.803, 57.054, 35.698, -51.409]
  Call Extruder(262.22712)
  MoveL 4471 to (239.78, 154.27, 69.25) mm, rotated rx 180 ry 0 rz 180 deg; joints [-29.343, 21.865, 46.786, 57.073, 35.719, -51.423]
  MoveL 4472 to (239.78, 154.27, 69.25) mm, rotated rx 180 ry 0 rz 180 deg; joints [-29.343, 21.865, 46.786, 57.073, 35.719, -51.423]
  Call Extruder(262.35848)
  MoveL 4473 to (239.71, 154.5, 69.25) mm, rotated rx 180 ry 0 rz 180 deg; joints [-29.366, 21.877, 46.77, 57.093, 35.74, -51.437]
  MoveL 4474 to (239.71, 154.5, 69.25) mm, rotated rx 180 ry 0 rz 180 deg; joints [-29.366, 21.877, 46.77, 57.093, 35.74, -51.437]
  Call Extruder(262.47038)
  MoveL 4475 to (239.65, 154.68, 69.25) mm, rotated rx -180 ry 0 rz -180 deg; joints [-29.386, 21.886, 46.757, 57.11, 35.758, -51.449]
  MoveL 4476 to (239.65, 154.68, 69.25) mm, rotated rx -180 ry 0 rz -180 deg; joints [-29.386, 21.886, 46.757, 57.11, 35.758, -51.449]
  Call Extruder(262.58272)
  MoveL 4477 to (239.59, 154.87, 69.25) mm, rotated rx 180 ry 0 rz 180 deg; joints [-29.406, 21.895, 46.744, 57.127, 35.775, -51.461]
  MoveL 4478 to (239.59, 154.87, 69.25) mm, rotated rx 180 ry 0 rz 180 deg; joints [-29.406, 21.895, 46.744, 57.127, 35.775, -51.461]
  Call Extruder(262.69551)
  MoveL 4479 to (239.53, 155.06, 69.25) mm, rotated rx 180 ry 0 rz -180 deg; joints [-29.426, 21.904, 46.732, 57.145, 35.793, -51.473]
  MoveL 4480 to (239.53, 155.06, 69.25) mm, rotated rx 180 ry 0 rz -180 deg; joints [-29.426, 21.904, 46.732, 57.145, 35.793, -51.473]
  Call Extruder(262.80875)
  MoveL 4481 to (239.47, 155.25, 69.25) mm, rotated rx 180 ry 0 rz 180 deg; joints [-29.446, 21.913, 46.719, 57.162, 35.81, -51.485]
  MoveL 4482 to (239.47, 155.25, 69.25) mm, rotated rx 180 ry 0 rz 180 deg; joints [-29.446, 21.913, 46.719, 57.162, 35.81, -51.485]
  Call Extruder(262.92243)
  MoveL 4483 to (239.41, 155.44, 69.25) mm, rotated rx -180 ry 0 rz 180 deg; joints [-29.466, 21.922, 46.706, 57.179, 35.828, -51.497]
  MoveL 4484 to (239.41, 155.44, 69.25) mm, rotated rx -180 ry 0 rz 180 deg; joints [-29.466, 21.922, 46.706, 57.179, 35.828, -51.497]
  Call Extruder(263.10439)
  MoveL 4485 to (239.29, 155.73, 69.25) mm, rotated rx 180 ry 0 rz 180 deg; joints [-29.499, 21.931, 46.694, 57.209, 35.855, -51.52]
  MoveL 4486 to (239.29, 155.73, 69.25) mm, rotated rx 180 ry 0 rz 180 deg; joints [-29.499, 21.931, 46.694, 57.209, 35.855, -51.52]
  Call Extruder(263.28710)
  MoveL 4487 to (239.16, 156.02, 69.25) mm, rotated rx -180 ry 0 rz -180 deg; joints [-29.531, 21.94, 46.681, 57.239, 35.883, -51.543]
  MoveL 4488 to (239.16, 156.02, 69.25) mm, rotated rx -180 ry 0 rz -180 deg; joints [-29.531, 21.94, 46.681, 57.239, 35.883, -51.543]
  Call Extruder(263.45752)
  MoveL 4489 to (239.05, 156.29, 69.25) mm, rotated rx 180 ry 0 rz 180 deg; joints [-29.561, 21.948, 46.67, 57.267, 35.908, -51.564]
  MoveL 4490 to (239.05, 156.29, 69.25) mm, rotated rx 180 ry 0 rz 180 deg; joints [-29.561, 21.948, 46.67, 57.267, 35.908, -51.564]
  Call Extruder(263.61554)
  MoveL 4491 to (238.94, 156.54, 69.25) mm, rotated rx 180 ry 0 rz 180 deg; joints [-29.589, 21.955, 46.661, 57.294, 35.931, -51.584]
  MoveL 4492 to (238.94, 156.54, 69.25) mm, rotated rx 180 ry 0 rz 180 deg; joints [-29.589, 21.955, 46.661, 57.294, 35.931, -51.584]
  Call Extruder(263.77415)
  MoveL 4493 to (238.84, 156.79, 69.25) mm, rotated rx -180 ry 0 rz 180 deg; joints [-29.617, 21.962, 46.651, 57.32, 35.954, -51.604]
  MoveL 4494 to (238.84, 156.79, 69.25) mm, rotated rx -180 ry 0 rz 180 deg; joints [-29.617, 21.962, 46.651, 57.32, 35.954, -51.604]
  Call Extruder(263.98032)
  MoveL 4495 to (238.66, 157.09, 69.25) mm, rotated rx 180 ry 0 rz 180 deg; joints [-29.653, 21.962, 46.651, 57.358, 35.983, -51.635]
  MoveL 4496 to (238.66, 157.09, 69.25) mm, rotated rx 180 ry 0 rz 180 deg; joints [-29.653, 21.962, 46.651, 57.358, 35.983, -51.635]
  Call Extruder(264.18727)
  MoveL 4497 to (238.49, 157.4, 69.25) mm, rotated rx -180 ry 0 rz 180 deg; joints [-29.689, 21.961, 46.652, 57.397, 36.011, -51.666]
  MoveL 4498 to (238.49, 157.4, 69.25) mm, rotated rx -180 ry 0 rz 180 deg; joints [-29.689, 21.961, 46.652, 57.397, 36.011, -51.666]
  Call Extruder(264.39499)
  MoveL 4499 to (238.31, 157.7, 69.25) mm, rotated rx -180 ry 0 rz 180 deg; joints [-29.725, 21.961, 46.653, 57.435, 36.039, -51.697]
  MoveL 4500 to (238.31, 157.7, 69.25) mm, rotated rx -180 ry 0 rz 180 deg; joints [-29.725, 21.961, 46.653, 57.435, 36.039, -51.697]
  Call Extruder(264.60350)
  MoveL 4501 to (238.13, 158.01, 69.25) mm, rotated rx -180 ry 0 rz 180 deg; joints [-29.761, 21.96, 46.653, 57.473, 36.067, -51.728]
  MoveL 4502 to (238.13, 158.01, 69.25) mm, rotated rx -180 ry 0 rz 180 deg; joints [-29.761, 21.96, 46.653, 57.473, 36.067, -51.728]
  Call Extruder(264.78304)
  MoveL 4503 to (237.96, 158.25, 69.25) mm, rotated rx -180 ry 0 rz 180 deg; joints [-29.792, 21.953, 46.663, 57.509, 36.09, -51.759]
  MoveL 4504 to (237.96, 158.25, 69.25) mm, rotated rx -180 ry 0 rz 180 deg; joints [-29.792, 21.953, 46.663, 57.509, 36.09, -51.759]
  Call Extruder(265.11645)
  MoveL 4505 to (237.63, 158.7, 69.25) mm, rotated rx 180 ry 0 rz -180 deg; joints [-29.849, 21.939, 46.683, 57.576, 36.132, -51.815]
  MoveL 4506 to (237.63, 158.7, 69.25) mm, rotated rx 180 ry 0 rz -180 deg; joints [-29.849, 21.939, 46.683, 57.576, 36.132, -51.815]
  Call Extruder(265.45104)
  MoveL 4507 to (237.3, 159.15, 69.25) mm, rotated rx 180 ry 0 rz 180 deg; joints [-29.907, 21.925, 46.702, 57.642, 36.174, -51.871]
  Call Extruder(266.27899)
  MoveL 4508 to (236.39, 160.19, 69.25) mm, rotated rx -180 ry 0 rz 180 deg; joints [-30.046, 21.862, 46.79, 57.816, 36.271, -52.025]
  Call Extruder(267.10694)
  MoveL 4509 to (235.35, 161.1, 69.25) mm, rotated rx 180 ry 0 rz -180 deg; joints [-30.182, 21.761, 46.932, 58.002, 36.356, -52.195]
  Call Extruder(267.27424)
  MoveL 4510 to (235.13, 161.27, 69.25) mm, rotated rx 180 ry 0 rz 180 deg; joints [-30.208, 21.735, 46.968, 58.042, 36.372, -52.231]
  MoveL 4511 to (235.13, 161.27, 69.25) mm, rotated rx 180 ry 0 rz 180 deg; joints [-30.208, 21.735, 46.968, 58.042, 36.372, -52.231]
  Call Extruder(267.60766)
  MoveL 4512 to (234.68, 161.6, 69.25) mm, rotated rx 180 ry 0 rz 180 deg; joints [-30.261, 21.683, 47.04, 58.119, 36.403, -52.304]
  MoveL 4513 to (234.68, 161.6, 69.25) mm, rotated rx 180 ry 0 rz 180 deg; joints [-30.261, 21.683, 47.04, 58.119, 36.403, -52.304]
  Call Extruder(267.93990)
  MoveL 4514 to (234.23, 161.92, 69.25) mm, rotated rx 180 ry 0 rz 180 deg; joints [-30.314, 21.631, 47.112, 58.197, 36.434, -52.377]
  MoveL 4515 to (234.23, 161.92, 69.25) mm, rotated rx 180 ry 0 rz 180 deg; joints [-30.314, 21.631, 47.112, 58.197, 36.434, -52.377]
  Call Extruder(268.05756)
  MoveL 4516 to (234.05, 162.02, 69.25) mm, rotated rx 180 ry 0 rz 180 deg; joints [-30.331, 21.609, 47.143, 58.225, 36.443, -52.404]
  MoveL 4517 to (234.05, 162.02, 69.25) mm, rotated rx 180 ry 0 rz 180 deg; joints [-30.331, 21.609, 47.143, 58.225, 36.443, -52.404]
  Call Extruder(268.26529)
  MoveL 4518 to (233.75, 162.2, 69.25) mm, rotated rx -180 ry 0 rz -180 deg; joints [-30.363, 21.569, 47.198, 58.275, 36.46, -52.452]
  MoveL 4519 to (233.75, 162.2, 69.25) mm, rotated rx -180 ry 0 rz -180 deg; joints [-30.363, 21.569, 47.198, 58.275, 36.46, -52.452]
  Call Extruder(268.47224)
  MoveL 4520 to (233.45, 162.37, 69.25) mm, rotated rx 180 ry 0 rz 180 deg; joints [-30.394, 21.529, 47.253, 58.326, 36.477, -52.5]
  MoveL 4521 to (233.45, 162.37, 69.25) mm, rotated rx 180 ry 0 rz 180 deg; joints [-30.394, 21.529, 47.253, 58.326, 36.477, -52.5]
  Call Extruder(268.67841)
  MoveL 4522 to (233.14, 162.55, 69.25) mm, rotated rx 180 ry 0 rz 180 deg; joints [-30.426, 21.489, 47.309, 58.376, 36.494, -52.548]
  MoveL 4523 to (233.14, 162.55, 69.25) mm, rotated rx 180 ry 0 rz 180 deg; joints [-30.426, 21.489, 47.309, 58.376, 36.494, -52.548]
  Call Extruder(268.86008)
  MoveL 4524 to (232.87, 162.69, 69.25) mm, rotated rx -180 ry 0 rz 180 deg; joints [-30.453, 21.451, 47.361, 58.42, 36.508, -52.592]
  MoveL 4525 to (232.87, 162.69, 69.25) mm, rotated rx -180 ry 0 rz 180 deg; joints [-30.453, 21.451, 47.361, 58.42, 36.508, -52.592]
  Call Extruder(269.01805)
  MoveL 4526 to (232.62, 162.8, 69.25) mm, rotated rx 180 ry 0 rz 180 deg; joints [-30.476, 21.415, 47.412, 58.46, 36.519, -52.631]
  MoveL 4527 to (232.62, 162.8, 69.25) mm, rotated rx 180 ry 0 rz 180 deg; joints [-30.476, 21.415, 47.412, 58.46, 36.519, -52.631]
  Call Extruder(269.17542)
  MoveL 4528 to (232.37, 162.91, 69.25) mm, rotated rx 180 ry 0 rz -180 deg; joints [-30.498, 21.378, 47.463, 58.499, 36.529, -52.669]
  MoveL 4529 to (232.37, 162.91, 69.25) mm, rotated rx 180 ry 0 rz -180 deg; joints [-30.498, 21.378, 47.463, 58.499, 36.529, -52.669]
  Call Extruder(269.35816)
  MoveL 4530 to (232.08, 163.03, 69.25) mm, rotated rx 180 ry 0 rz 180 deg; joints [-30.524, 21.335, 47.523, 58.545, 36.541, -52.715]
  MoveL 4531 to (232.08, 163.03, 69.25) mm, rotated rx 180 ry 0 rz 180 deg; joints [-30.524, 21.335, 47.523, 58.545, 36.541, -52.715]
  Call Extruder(269.54014)
  MoveL 4532 to (231.78, 163.15, 69.25) mm, rotated rx -180 ry 0 rz 180 deg; joints [-30.551, 21.291, 47.583, 58.591, 36.553, -52.76]
  MoveL 4533 to (231.78, 163.15, 69.25) mm, rotated rx -180 ry 0 rz 180 deg; joints [-30.551, 21.291, 47.583, 58.591, 36.553, -52.76]
  Call Extruder(269.68748)
  MoveL 4534 to (231.54, 163.24, 69.25) mm, rotated rx 180 ry 0 rz 180 deg; joints [-30.571, 21.255, 47.633, 58.628, 36.563, -52.797]
  MoveL 4535 to (231.54, 163.24, 69.25) mm, rotated rx 180 ry 0 rz 180 deg; joints [-30.571, 21.255, 47.633, 58.628, 36.563, -52.797]
  Call Extruder(269.80071)
  MoveL 4536 to (231.35, 163.3, 69.25) mm, rotated rx 180 ry 0 rz 180 deg; joints [-30.587, 21.225, 47.675, 58.657, 36.569, -52.826]
  MoveL 4537 to (231.35, 163.3, 69.25) mm, rotated rx 180 ry 0 rz 180 deg; joints [-30.587, 21.225, 47.675, 58.657, 36.569, -52.826]
  Call Extruder(269.91348)
  MoveL 4538 to (231.17, 163.36, 69.25) mm, rotated rx 180 ry 0 rz 180 deg; joints [-30.602, 21.195, 47.716, 58.685, 36.575, -52.855]
  MoveL 4539 to (231.17, 163.36, 69.25) mm, rotated rx 180 ry 0 rz 180 deg; joints [-30.602, 21.195, 47.716, 58.685, 36.575, -52.855]
  Call Extruder(270.02582)
  MoveL 4540 to (230.98, 163.42, 69.25) mm, rotated rx 180 ry 0 rz -180 deg; joints [-30.618, 21.166, 47.757, 58.714, 36.582, -52.884]
  MoveL 4541 to (230.98, 163.42, 69.25) mm, rotated rx 180 ry 0 rz -180 deg; joints [-30.618, 21.166, 47.757, 58.714, 36.582, -52.884]
  Call Extruder(270.13770)
  MoveL 4542 to (230.79, 163.48, 69.25) mm, rotated rx 180 ry 0 rz -180 deg; joints [-30.633, 21.136, 47.798, 58.743, 36.588, -52.912]
  MoveL 4543 to (230.79, 163.48, 69.25) mm, rotated rx 180 ry 0 rz -180 deg; joints [-30.633, 21.136, 47.798, 58.743, 36.588, -52.912]
  Call Extruder(270.25911)
  MoveL 4544 to (230.58, 163.55, 69.25) mm, rotated rx 180 ry 0 rz 180 deg; joints [-30.65, 21.103, 47.843, 58.774, 36.595, -52.944]
  MoveL 4545 to (230.58, 163.55, 69.25) mm, rotated rx 180 ry 0 rz 180 deg; joints [-30.65, 21.103, 47.843, 58.774, 36.595, -52.944]
  Call Extruder(270.38992)
  MoveL 4546 to (230.36, 163.61, 69.25) mm, rotated rx -180 ry 0 rz 180 deg; joints [-30.668, 21.068, 47.892, 58.808, 36.602, -52.978]
  MoveL 4547 to (230.36, 163.61, 69.25) mm, rotated rx -180 ry 0 rz 180 deg; joints [-30.668, 21.068, 47.892, 58.808, 36.602, -52.978]
  Call Extruder(270.52017)
  MoveL 4548 to (230.14, 163.68, 69.25) mm, rotated rx 180 ry 0 rz -180 deg; joints [-30.685, 21.032, 47.941, 58.841, 36.61, -53.011]
  MoveL 4549 to (230.14, 163.68, 69.25) mm, rotated rx 180 ry 0 rz -180 deg; joints [-30.685, 21.032, 47.941, 58.841, 36.61, -53.011]
  Call Extruder(270.64985)
  MoveL 4550 to (229.91, 163.75, 69.25) mm, rotated rx 180 ry 0 rz 180 deg; joints [-30.703, 20.996, 47.99, 58.875, 36.617, -53.045]
  MoveL 4551 to (229.91, 163.75, 69.25) mm, rotated rx 180 ry 0 rz 180 deg; joints [-30.703, 20.996, 47.99, 58.875, 36.617, -53.045]
  Call Extruder(270.77897)
  MoveL 4552 to (229.69, 163.82, 69.25) mm, rotated rx -180 ry 0 rz 180 deg; joints [-30.721, 20.961, 48.04, 58.908, 36.624, -53.079]
  MoveL 4553 to (229.69, 163.82, 69.25) mm, rotated rx -180 ry 0 rz 180 deg; joints [-30.721, 20.961, 48.04, 58.908, 36.624, -53.079]
  Call Extruder(270.89404)
  MoveL 4554 to (229.48, 163.86, 69.25) mm, rotated rx 180 ry 0 rz 180 deg; joints [-30.736, 20.926, 48.087, 58.938, 36.629, -53.11]
  MoveL 4555 to (229.48, 163.86, 69.25) mm, rotated rx 180 ry 0 rz 180 deg; joints [-30.736, 20.926, 48.087, 58.938, 36.629, -53.11]
  Call Extruder(271.00867)
  MoveL 4556 to (229.28, 163.91, 69.25) mm, rotated rx -180 ry 0 rz 180 deg; joints [-30.751, 20.892, 48.134, 58.968, 36.635, -53.14]
  MoveL 4557 to (229.28, 163.91, 69.25) mm, rotated rx -180 ry 0 rz 180 deg; joints [-30.751, 20.892, 48.134, 58.968, 36.635, -53.14]
  Call Extruder(271.12284)
  MoveL 4558 to (229.08, 163.95, 69.25) mm, rotated rx -180 ry 0 rz -180 deg; joints [-30.766, 20.858, 48.181, 58.998, 36.64, -53.171]
  MoveL 4559 to (229.08, 163.95, 69.25) mm, rotated rx -180 ry 0 rz -180 deg; joints [-30.766, 20.858, 48.181, 58.998, 36.64, -53.171]
  Call Extruder(271.23656)
  MoveL 4560 to (228.87, 164, 69.25) mm, rotated rx 180 ry 0 rz -180 deg; joints [-30.781, 20.823, 48.229, 59.028, 36.645, -53.201]
  MoveL 4561 to (228.87, 164, 69.25) mm, rotated rx 180 ry 0 rz -180 deg; joints [-30.781, 20.823, 48.229, 59.028, 36.645, -53.201]
  Call Extruder(271.36198)
  MoveL 4562 to (228.64, 164.04, 69.25) mm, rotated rx 180 ry 0 rz 180 deg; joints [-30.797, 20.785, 48.281, 59.06, 36.651, -53.235]
  MoveL 4563 to (228.64, 164.04, 69.25) mm, rotated rx 180 ry 0 rz 180 deg; joints [-30.797, 20.785, 48.281, 59.06, 36.651, -53.235]
  Call Extruder(271.49895)
  MoveL 4564 to (228.4, 164.09, 69.25) mm, rotated rx 180 ry 0 rz 180 deg; joints [-30.815, 20.743, 48.339, 59.096, 36.657, -53.272]
  MoveL 4565 to (228.4, 164.09, 69.25) mm, rotated rx 180 ry 0 rz 180 deg; joints [-30.815, 20.743, 48.339, 59.096, 36.657, -53.272]
  Call Extruder(271.63532)
  MoveL 4566 to (228.15, 164.14, 69.25) mm, rotated rx 180 ry 0 rz 180 deg; joints [-30.832, 20.701, 48.397, 59.132, 36.663, -53.309]
  MoveL 4567 to (228.15, 164.14, 69.25) mm, rotated rx 180 ry 0 rz 180 deg; joints [-30.832, 20.701, 48.397, 59.132, 36.663, -53.309]
  Call Extruder(271.77108)
  MoveL 4568 to (227.9, 164.19, 69.25) mm, rotated rx 180 ry 0 rz -180 deg; joints [-30.85, 20.659, 48.455, 59.168, 36.669, -53.345]
  MoveL 4569 to (227.9, 164.19, 69.25) mm, rotated rx 180 ry 0 rz -180 deg; joints [-30.85, 20.659, 48.455, 59.168, 36.669, -53.345]
  Call Extruder(271.90623)
  MoveL 4570 to (227.65, 164.24, 69.25) mm, rotated rx -180 ry 0 rz 180 deg; joints [-30.868, 20.617, 48.513, 59.204, 36.675, -53.382]
  MoveL 4571 to (227.65, 164.24, 69.25) mm, rotated rx -180 ry 0 rz 180 deg; joints [-30.868, 20.617, 48.513, 59.204, 36.675, -53.382]
  Call Extruder(272.04076)
  MoveL 4572 to (227.4, 164.29, 69.25) mm, rotated rx 180 ry 0 rz 180 deg; joints [-30.886, 20.575, 48.57, 59.239, 36.682, -53.419]
  MoveL 4573 to (227.4, 164.29, 69.25) mm, rotated rx 180 ry 0 rz 180 deg; joints [-30.886, 20.575, 48.57, 59.239, 36.682, -53.419]
  Call Extruder(272.17469)
  MoveL 4574 to (227.15, 164.34, 69.25) mm, rotated rx -180 ry 0 rz 180 deg; joints [-30.903, 20.533, 48.627, 59.275, 36.688, -53.455]
  MoveL 4575 to (227.15, 164.34, 69.25) mm, rotated rx -180 ry 0 rz 180 deg; joints [-30.903, 20.533, 48.627, 59.275, 36.688, -53.455]
  Call Extruder(272.32256)
  MoveL 4576 to (226.87, 164.39, 69.25) mm, rotated rx -180 ry 0 rz 180 deg; joints [-30.923, 20.485, 48.692, 59.314, 36.695, -53.496]
  MoveL 4577 to (226.87, 164.39, 69.25) mm, rotated rx -180 ry 0 rz 180 deg; joints [-30.923, 20.485, 48.692, 59.314, 36.695, -53.496]
  Call Extruder(272.48429)
  MoveL 4578 to (226.57, 164.44, 69.25) mm, rotated rx 180 ry 0 rz 180 deg; joints [-30.943, 20.433, 48.764, 59.357, 36.701, -53.54]
  MoveL 4579 to (226.57, 164.44, 69.25) mm, rotated rx 180 ry 0 rz 180 deg; joints [-30.943, 20.433, 48.764, 59.357, 36.701, -53.54]
  Call Extruder(272.64531)
  MoveL 4580 to (226.26, 164.49, 69.25) mm, rotated rx -180 ry 0 rz 180 deg; joints [-30.964, 20.38, 48.836, 59.4, 36.708, -53.584]
  MoveL 4581 to (226.26, 164.49, 69.25) mm, rotated rx -180 ry 0 rz 180 deg; joints [-30.964, 20.38, 48.836, 59.4, 36.708, -53.584]
  Call Extruder(272.80559)
  MoveL 4582 to (225.95, 164.54, 69.25) mm, rotated rx 180 ry 0 rz 180 deg; joints [-30.985, 20.328, 48.908, 59.443, 36.715, -53.629]
  MoveL 4583 to (225.95, 164.54, 69.25) mm, rotated rx 180 ry 0 rz 180 deg; joints [-30.985, 20.328, 48.908, 59.443, 36.715, -53.629]
  Call Extruder(272.96514)
  MoveL 4584 to (225.65, 164.58, 69.25) mm, rotated rx -180 ry 0 rz -180 deg; joints [-31.006, 20.275, 48.979, 59.486, 36.722, -53.673]
  MoveL 4585 to (225.65, 164.58, 69.25) mm, rotated rx -180 ry 0 rz -180 deg; joints [-31.006, 20.275, 48.979, 59.486, 36.722, -53.673]
  Call Extruder(273.12397)
  MoveL 4586 to (225.34, 164.63, 69.25) mm, rotated rx 180 ry 0 rz -180 deg; joints [-31.027, 20.223, 49.051, 59.528, 36.729, -53.717]
  MoveL 4587 to (225.34, 164.63, 69.25) mm, rotated rx 180 ry 0 rz -180 deg; joints [-31.027, 20.223, 49.051, 59.528, 36.729, -53.717]
  Call Extruder(273.30264)
  MoveL 4588 to (225, 164.68, 69.25) mm, rotated rx 180 ry 0 rz 180 deg; joints [-31.049, 20.163, 49.133, 59.576, 36.737, -53.766]
  MoveL 4589 to (225, 164.68, 69.25) mm, rotated rx 180 ry 0 rz 180 deg; joints [-31.049, 20.163, 49.133, 59.576, 36.737, -53.766]
  Call Extruder(273.50108)
  MoveL 4590 to (224.61, 164.72, 69.25) mm, rotated rx 180 ry 0 rz -180 deg; joints [-31.074, 20.095, 49.225, 59.629, 36.744, -53.822]
  MoveL 4591 to (224.61, 164.72, 69.25) mm, rotated rx 180 ry 0 rz -180 deg; joints [-31.074, 20.095, 49.225, 59.629, 36.744, -53.822]
  Call Extruder(273.69866)
  MoveL 4592 to (224.22, 164.77, 69.25) mm, rotated rx 180 ry 0 rz 180 deg; joints [-31.1, 20.027, 49.317, 59.682, 36.752, -53.877]
  MoveL 4593 to (224.22, 164.77, 69.25) mm, rotated rx 180 ry 0 rz 180 deg; joints [-31.1, 20.027, 49.317, 59.682, 36.752, -53.877]
  Call Extruder(273.89536)
  MoveL 4594 to (223.83, 164.82, 69.25) mm, rotated rx 180 ry 0 rz 180 deg; joints [-31.125, 19.96, 49.409, 59.735, 36.76, -53.931]
  MoveL 4595 to (223.83, 164.82, 69.25) mm, rotated rx 180 ry 0 rz 180 deg; joints [-31.125, 19.96, 49.409, 59.735, 36.76, -53.931]
  Call Extruder(274.09120)
  MoveL 4596 to (223.45, 164.86, 69.25) mm, rotated rx -180 ry 0 rz 180 deg; joints [-31.15, 19.892, 49.501, 59.788, 36.769, -53.986]
  MoveL 4597 to (223.45, 164.86, 69.25) mm, rotated rx -180 ry 0 rz 180 deg; joints [-31.15, 19.892, 49.501, 59.788, 36.769, -53.986]
  Call Extruder(274.38656)
  MoveL 4598 to (222.86, 164.91, 69.25) mm, rotated rx -180 ry 0 rz -180 deg; joints [-31.186, 19.788, 49.643, 59.866, 36.779, -54.068]
  MoveL 4599 to (222.86, 164.91, 69.25) mm, rotated rx -180 ry 0 rz -180 deg; joints [-31.186, 19.788, 49.643, 59.866, 36.779, -54.068]
  Call Extruder(274.68059)
  MoveL 4600 to (222.27, 164.96, 69.25) mm, rotated rx 180 ry 0 rz 180 deg; joints [-31.222, 19.683, 49.784, 59.944, 36.79, -54.15]
  MoveL 4601 to (222.27, 164.96, 69.25) mm, rotated rx 180 ry 0 rz 180 deg; joints [-31.222, 19.683, 49.784, 59.944, 36.79, -54.15]
  Call Extruder(274.97329)
  MoveL 4602 to (221.68, 165, 69.25) mm, rotated rx -180 ry 0 rz 180 deg; joints [-31.258, 19.579, 49.925, 60.022, 36.801, -54.232]
  MoveL 4603 to (221.68, 165, 69.25) mm, rotated rx -180 ry 0 rz 180 deg; joints [-31.258, 19.579, 49.925, 60.022, 36.801, -54.232]
  Call Extruder(275.54673)
  MoveL 4604 to (220.52, 165.05, 69.25) mm, rotated rx 180 ry 0 rz 180 deg; joints [-31.326, 19.37, 50.208, 60.173, 36.819, -54.39]
  MoveL 4605 to (220.52, 165.05, 69.25) mm, rotated rx 180 ry 0 rz 180 deg; joints [-31.326, 19.37, 50.208, 60.173, 36.819, -54.39]
  Call Extruder(276.26074)
  MoveL 4606 to (219.06, 165.09, 69.25) mm, rotated rx 180 ry 0 rz 180 deg; joints [-31.409, 19.107, 50.561, 60.359, 36.842, -54.586]
  Call Extruder(393.10748)
  MoveL 4607 to (-19.06, 165.09, 69.25) mm, rotated rx 180 ry 0 rz 180 deg; joints [-51.475, -11.065, 82.897, 76.059, 53.715, -67.244]
  Call Extruder(393.53608)
  MoveL 4608 to (-19.94, 165.07, 69.25) mm, rotated rx -180 ry 0 rz 180 deg; joints [-51.582, -11.145, 82.962, 76.099, 53.817, -67.255]
  MoveL 4609 to (-19.94, 165.07, 69.25) mm, rotated rx -180 ry 0 rz 180 deg; joints [-51.582, -11.145, 82.962, 76.099, 53.817, -67.255]
  Call Extruder(394.10954)
  MoveL 4610 to (-21.1, 165.03, 69.25) mm, rotated rx 180 ry 0 rz -180 deg; joints [-51.722, -11.253, 83.048, 76.151, 53.952, -67.269]
  MoveL 4611 to (-21.1, 165.03, 69.25) mm, rotated rx 180 ry 0 rz -180 deg; joints [-51.722, -11.253, 83.048, 76.151, 53.952, -67.269]
  Call Extruder(394.54383)
  MoveL 4612 to (-21.97, 164.98, 69.25) mm, rotated rx 180 ry 0 rz 180 deg; joints [-51.827, -11.336, 83.114, 76.189, 54.053, -67.279]
  MoveL 4613 to (-21.97, 164.98, 69.25) mm, rotated rx 180 ry 0 rz 180 deg; joints [-51.827, -11.336, 83.114, 76.189, 54.053, -67.279]
  Call Extruder(394.83786)
  MoveL 4614 to (-22.56, 164.93, 69.25) mm, rotated rx 180 ry 0 rz -180 deg; joints [-51.897, -11.393, 83.16, 76.214, 54.119, -67.284]
  MoveL 4615 to (-22.56, 164.93, 69.25) mm, rotated rx 180 ry 0 rz -180 deg; joints [-51.897, -11.393, 83.16, 76.214, 54.119, -67.284]
  Call Extruder(395.13322)
  MoveL 4616 to (-23.15, 164.89, 69.25) mm, rotated rx -180 ry 0 rz 180 deg; joints [-51.966, -11.45, 83.206, 76.239, 54.186, -67.29]
  MoveL 4617 to (-23.15, 164.89, 69.25) mm, rotated rx -180 ry 0 rz 180 deg; joints [-51.966, -11.45, 83.206, 76.239, 54.186, -67.29]
  Call Extruder(395.37944)
  MoveL 4618 to (-23.64, 164.84, 69.25) mm, rotated rx 180 ry 0 rz 180 deg; joints [-52.023, -11.498, 83.244, 76.259, 54.241, -67.294]
  MoveL 4619 to (-23.64, 164.84, 69.25) mm, rotated rx 180 ry 0 rz 180 deg; joints [-52.023, -11.498, 83.244, 76.259, 54.241, -67.294]
  Call Extruder(395.57615)
  MoveL 4620 to (-24.03, 164.79, 69.25) mm, rotated rx 180 ry 0 rz 180 deg; joints [-52.067, -11.538, 83.275, 76.275, 54.284, -67.296]
  MoveL 4621 to (-24.03, 164.79, 69.25) mm, rotated rx 180 ry 0 rz 180 deg; joints [-52.067, -11.538, 83.275, 76.275, 54.284, -67.296]
  Call Extruder(395.77372)
  MoveL 4622 to (-24.42, 164.75, 69.25) mm, rotated rx 180 ry 0 rz 180 deg; joints [-52.112, -11.577, 83.306, 76.29, 54.326, -67.299]
  MoveL 4623 to (-24.42, 164.75, 69.25) mm, rotated rx 180 ry 0 rz 180 deg; joints [-52.112, -11.577, 83.306, 76.29, 54.326, -67.299]
  Call Extruder(395.97216)
  MoveL 4624 to (-24.8, 164.7, 69.25) mm, rotated rx -180 ry 0 rz 180 deg; joints [-52.156, -11.616, 83.338, 76.306, 54.369, -67.302]
  MoveL 4625 to (-24.8, 164.7, 69.25) mm, rotated rx -180 ry 0 rz 180 deg; joints [-52.156, -11.616, 83.338, 76.306, 54.369, -67.302]
  Call Extruder(396.17147)
  MoveL 4626 to (-25.19, 164.66, 69.25) mm, rotated rx -180 ry 0 rz -180 deg; joints [-52.2, -11.655, 83.369, 76.321, 54.412, -67.304]
  MoveL 4627 to (-25.19, 164.66, 69.25) mm, rotated rx -180 ry 0 rz -180 deg; joints [-52.2, -11.655, 83.369, 76.321, 54.412, -67.304]
  Call Extruder(396.33030)
  MoveL 4628 to (-25.5, 164.61, 69.25) mm, rotated rx 180 ry 0 rz 180 deg; joints [-52.235, -11.687, 83.394, 76.333, 54.445, -67.306]
  MoveL 4629 to (-25.5, 164.61, 69.25) mm, rotated rx 180 ry 0 rz 180 deg; joints [-52.235, -11.687, 83.394, 76.333, 54.445, -67.306]
  Call Extruder(396.48986)
  MoveL 4630 to (-25.8, 164.56, 69.25) mm, rotated rx 180 ry 0 rz 180 deg; joints [-52.269, -11.72, 83.42, 76.344, 54.478, -67.307]
  MoveL 4631 to (-25.8, 164.56, 69.25) mm, rotated rx 180 ry 0 rz 180 deg; joints [-52.269, -11.72, 83.42, 76.344, 54.478, -67.307]
  Call Extruder(396.65015)
  MoveL 4632 to (-26.11, 164.51, 69.25) mm, rotated rx 180 ry 0 rz 180 deg; joints [-52.303, -11.752, 83.445, 76.356, 54.511, -67.309]
  MoveL 4633 to (-26.11, 164.51, 69.25) mm, rotated rx 180 ry 0 rz 180 deg; joints [-52.303, -11.752, 83.445, 76.356, 54.511, -67.309]
  Call Extruder(396.81116)
  MoveL 4634 to (-26.41, 164.46, 69.25) mm, rotated rx -180 ry 0 rz 180 deg; joints [-52.337, -11.784, 83.47, 76.367, 54.544, -67.31]
  MoveL 4635 to (-26.41, 164.46, 69.25) mm, rotated rx -180 ry 0 rz 180 deg; joints [-52.337, -11.784, 83.47, 76.367, 54.544, -67.31]
  Call Extruder(396.97291)
  MoveL 4636 to (-26.72, 164.41, 69.25) mm, rotated rx 180 ry 0 rz -180 deg; joints [-52.371, -11.816, 83.496, 76.379, 54.577, -67.311]
  MoveL 4637 to (-26.72, 164.41, 69.25) mm, rotated rx 180 ry 0 rz -180 deg; joints [-52.371, -11.816, 83.496, 76.379, 54.577, -67.311]
  Call Extruder(397.13538)
  MoveL 4638 to (-27.03, 164.37, 69.25) mm, rotated rx 180 ry 0 rz 180 deg; joints [-52.405, -11.848, 83.521, 76.39, 54.61, -67.313]
  MoveL 4639 to (-27.03, 164.37, 69.25) mm, rotated rx 180 ry 0 rz 180 deg; joints [-52.405, -11.848, 83.521, 76.39, 54.61, -67.313]
  Call Extruder(397.26930)
  MoveL 4640 to (-27.27, 164.32, 69.25) mm, rotated rx 180 ry 0 rz 180 deg; joints [-52.432, -11.875, 83.543, 76.399, 54.637, -67.313]
  MoveL 4641 to (-27.27, 164.32, 69.25) mm, rotated rx 180 ry 0 rz 180 deg; joints [-52.432, -11.875, 83.543, 76.399, 54.637, -67.313]
  Call Extruder(397.40384)
  MoveL 4642 to (-27.52, 164.27, 69.25) mm, rotated rx 180 ry 0 rz 180 deg; joints [-52.459, -11.902, 83.564, 76.408, 54.663, -67.314]
  MoveL 4643 to (-27.52, 164.27, 69.25) mm, rotated rx 180 ry 0 rz 180 deg; joints [-52.459, -11.902, 83.564, 76.408, 54.663, -67.314]
  Call Extruder(397.53899)
  MoveL 4644 to (-27.77, 164.22, 69.25) mm, rotated rx -180 ry 0 rz 180 deg; joints [-52.486, -11.93, 83.586, 76.417, 54.689, -67.314]
  MoveL 4645 to (-27.77, 164.22, 69.25) mm, rotated rx -180 ry 0 rz 180 deg; joints [-52.486, -11.93, 83.586, 76.417, 54.689, -67.314]
  Call Extruder(397.67474)
  MoveL 4646 to (-28.02, 164.17, 69.25) mm, rotated rx 180 ry 0 rz -180 deg; joints [-52.513, -11.957, 83.607, 76.425, 54.715, -67.315]
  MoveL 4647 to (-28.02, 164.17, 69.25) mm, rotated rx 180 ry 0 rz -180 deg; joints [-52.513, -11.957, 83.607, 76.425, 54.715, -67.315]
  Call Extruder(397.81111)
  MoveL 4648 to (-28.27, 164.12, 69.25) mm, rotated rx 180 ry 0 rz 180 deg; joints [-52.54, -11.984, 83.628, 76.434, 54.742, -67.315]
  MoveL 4649 to (-28.27, 164.12, 69.25) mm, rotated rx 180 ry 0 rz 180 deg; joints [-52.54, -11.984, 83.628, 76.434, 54.742, -67.315]
  Call Extruder(397.89597)
  MoveL 4650 to (-28.43, 164.09, 69.25) mm, rotated rx -180 ry 0 rz 180 deg; joints [-52.556, -12.001, 83.642, 76.44, 54.758, -67.316]
  Set speed (130.0 mm/s)
  MoveL 4651 to (-31.76, 163.31, 69.25) mm, rotated rx 180 ry 0 rz 180 deg; joints [-52.91, -12.376, 83.935, 76.551, 55.103, -67.315]
  MoveL 4652 to (-31.76, 163.31, 78.65) mm, rotated rx -180 ry 0 rz 180 deg; joints [-52.91, -13.157, 86.045, 77.459, 54.804, -68.896]
  Call Extruder(395.89597)
  Set speed (40.0 mm/s)
  MoveL 4653 to (-31.76, 163.31, 78.65) mm, rotated rx -180 ry 0 rz 180 deg; joints [-52.91, -13.157, 86.045, 77.459, 54.804, -68.896]
  Call Extruder(0.00000)
  Set speed (130.0 mm/s)
  MoveL 4654 to (-31.64, 163.21, 78.65) mm, rotated rx -180 ry 0 rz -180 deg; joints [-52.884, -13.158, 86.046, 77.447, 54.78, -68.889]
  Call Extruder(2.00000)
  Set speed (40.0 mm/s)
  MoveL 4655 to (-31.64, 163.21, 78.65) mm, rotated rx -180 ry 0 rz -180 deg; joints [-52.884, -13.158, 86.046, 77.447, 54.78, -68.889]
  Set speed (30.0 mm/s)
  MoveL 4656 to (-31.64, 163.21, 78.65) mm, rotated rx -180 ry 0 rz -180 deg; joints [-52.884, -13.158, 86.046, 77.447, 54.78, -68.889]
  Call Extruder(2.18198)
  MoveL 4657 to (-31.93, 163.09, 78.65) mm, rotated rx -180 ry 0 rz -180 deg; joints [-52.91, -13.197, 86.076, 77.452, 54.806, -68.885]
  MoveL 4658 to (-31.93, 163.09, 78.65) mm, rotated rx -180 ry 0 rz -180 deg; joints [-52.91, -13.197, 86.076, 77.452, 54.806, -68.885]
  Call Extruder(2.36471)
  MoveL 4659 to (-32.22, 162.97, 78.65) mm, rotated rx 180 ry 0 rz 180 deg; joints [-52.936, -13.236, 86.106, 77.458, 54.833, -68.881]
  MoveL 4660 to (-32.22, 162.97, 78.65) mm, rotated rx 180 ry 0 rz 180 deg; joints [-52.936, -13.236, 86.106, 77.458, 54.833, -68.881]
  Call Extruder(2.53513)
  MoveL 4661 to (-32.49, 162.85, 78.65) mm, rotated rx 180 ry 0 rz 180 deg; joints [-52.96, -13.272, 86.133, 77.463, 54.857, -68.877]
  MoveL 4662 to (-32.49, 162.85, 78.65) mm, rotated rx 180 ry 0 rz 180 deg; joints [-52.96, -13.272, 86.133, 77.463, 54.857, -68.877]
  Call Extruder(2.69310)
  MoveL 4663 to (-32.74, 162.74, 78.65) mm, rotated rx -180 ry 0 rz 180 deg; joints [-52.982, -13.305, 86.159, 77.467, 54.879, -68.873]
  MoveL 4664 to (-32.74, 162.74, 78.65) mm, rotated rx -180 ry 0 rz 180 deg; joints [-52.982, -13.305, 86.159, 77.467, 54.879, -68.873]
  Call Extruder(2.85168)
  MoveL 4665 to (-32.99, 162.64, 78.65) mm, rotated rx 180 ry 0 rz 180 deg; joints [-53.004, -13.339, 86.185, 77.471, 54.901, -68.869]
  MoveL 4666 to (-32.99, 162.64, 78.65) mm, rotated rx 180 ry 0 rz 180 deg; joints [-53.004, -13.339, 86.185, 77.471, 54.901, -68.869]
  Call Extruder(3.05784)
  MoveL 4667 to (-33.29, 162.46, 78.65) mm, rotated rx 180 ry 0 rz 180 deg; joints [-53.026, -13.385, 86.22, 77.474, 54.924, -68.862]
  MoveL 4668 to (-33.29, 162.46, 78.65) mm, rotated rx 180 ry 0 rz 180 deg; joints [-53.026, -13.385, 86.22, 77.474, 54.924, -68.862]
  Call Extruder(3.26479)
  MoveL 4669 to (-33.6, 162.29, 78.65) mm, rotated rx 180 ry 0 rz 180 deg; joints [-53.049, -13.431, 86.255, 77.476, 54.947, -68.855]
  MoveL 4670 to (-33.6, 162.29, 78.65) mm, rotated rx 180 ry 0 rz 180 deg; joints [-53.049, -13.431, 86.255, 77.476, 54.947, -68.855]
  Call Extruder(3.47251)
  MoveL 4671 to (-33.9, 162.11, 78.65) mm, rotated rx 180 ry 0 rz 180 deg; joints [-53.071, -13.477, 86.29, 77.479, 54.971, -68.848]
  MoveL 4672 to (-33.9, 162.11, 78.65) mm, rotated rx 180 ry 0 rz 180 deg; joints [-53.071, -13.477, 86.29, 77.479, 54.971, -68.848]
  Call Extruder(3.68102)
  MoveL 4673 to (-34.21, 161.94, 78.65) mm, rotated rx 180 ry 0 rz 180 deg; joints [-53.094, -13.522, 86.325, 77.481, 54.994, -68.841]
  MoveL 4674 to (-34.21, 161.94, 78.65) mm, rotated rx 180 ry 0 rz 180 deg; joints [-53.094, -13.522, 86.325, 77.481, 54.994, -68.841]
  Call Extruder(3.86055)
  MoveL 4675 to (-34.45, 161.76, 78.65) mm, rotated rx 180 ry 0 rz 180 deg; joints [-53.109, -13.563, 86.356, 77.481, 55.01, -68.833]
  MoveL 4676 to (-34.45, 161.76, 78.65) mm, rotated rx 180 ry 0 rz 180 deg; joints [-53.109, -13.563, 86.356, 77.481, 55.01, -68.833]
  Call Extruder(4.19399)
  MoveL 4677 to (-34.9, 161.43, 78.65) mm, rotated rx 180 ry 0 rz 180 deg; joints [-53.135, -13.639, 86.414, 77.481, 55.039, -68.818]
  MoveL 4678 to (-34.9, 161.43, 78.65) mm, rotated rx 180 ry 0 rz 180 deg; joints [-53.135, -13.639, 86.414, 77.481, 55.039, -68.818]
  Call Extruder(4.52861)
  MoveL 4679 to (-35.35, 161.1, 78.65) mm, rotated rx -180 ry 0 rz 180 deg; joints [-53.163, -13.715, 86.471, 77.48, 55.068, -68.803]
  Call Extruder(5.35652)
  MoveL 4680 to (-36.39, 160.19, 78.65) mm, rotated rx -180 ry 0 rz 180 deg; joints [-53.209, -13.906, 86.617, 77.469, 55.122, -68.76]
  Call Extruder(6.18445)
  MoveL 4681 to (-37.3, 159.15, 78.65) mm, rotated rx 180 ry 0 rz 180 deg; joints [-53.227, -14.101, 86.764, 77.445, 55.149, -68.708]
  Call Extruder(6.35176)
  MoveL 4682 to (-37.47, 158.93, 78.65) mm, rotated rx -180 ry 0 rz 180 deg; joints [-53.227, -14.14, 86.793, 77.438, 55.151, -68.696]
  MoveL 4683 to (-37.47, 158.93, 78.65) mm, rotated rx -180 ry 0 rz 180 deg; joints [-53.227, -14.14, 86.793, 77.438, 55.151, -68.696]
  Call Extruder(6.68519)
  MoveL 4684 to (-37.8, 158.48, 78.65) mm, rotated rx -180 ry 0 rz 180 deg; joints [-53.226, -14.219, 86.853, 77.424, 55.154, -68.672]
  MoveL 4685 to (-37.8, 158.48, 78.65) mm, rotated rx -180 ry 0 rz 180 deg; joints [-53.226, -14.219, 86.853, 77.424, 55.154, -68.672]
  Call Extruder(7.01743)
  MoveL 4686 to (-38.12, 158.02, 78.65) mm, rotated rx 180 ry 0 rz -180 deg; joints [-53.224, -14.298, 86.912, 77.41, 55.157, -68.649]
  MoveL 4687 to (-38.12, 158.02, 78.65) mm, rotated rx 180 ry 0 rz -180 deg; joints [-53.224, -14.298, 86.912, 77.41, 55.157, -68.649]
  Call Extruder(7.13511)
  MoveL 4688 to (-38.22, 157.85, 78.65) mm, rotated rx 180 ry 0 rz 180 deg; joints [-53.221, -14.326, 86.933, 77.404, 55.155, -68.639]
  MoveL 4689 to (-38.22, 157.85, 78.65) mm, rotated rx 180 ry 0 rz 180 deg; joints [-53.221, -14.326, 86.933, 77.404, 55.155, -68.639]
  Call Extruder(7.34283)
  MoveL 4690 to (-38.4, 157.55, 78.65) mm, rotated rx -180 ry 0 rz 180 deg; joints [-53.214, -14.375, 86.97, 77.392, 55.151, -68.623]
  MoveL 4691 to (-38.4, 157.55, 78.65) mm, rotated rx -180 ry 0 rz 180 deg; joints [-53.214, -14.375, 86.97, 77.392, 55.151, -68.623]
  Call Extruder(7.54978)
  MoveL 4692 to (-38.57, 157.25, 78.65) mm, rotated rx 180 ry 0 rz 180 deg; joints [-53.207, -14.424, 87.006, 77.381, 55.147, -68.606]
  MoveL 4693 to (-38.57, 157.25, 78.65) mm, rotated rx 180 ry 0 rz 180 deg; joints [-53.207, -14.424, 87.006, 77.381, 55.147, -68.606]
  Call Extruder(7.75595)
  MoveL 4694 to (-38.75, 156.94, 78.65) mm, rotated rx 180 ry 0 rz 180 deg; joints [-53.2, -14.474, 87.043, 77.369, 55.144, -68.59]
  MoveL 4695 to (-38.75, 156.94, 78.65) mm, rotated rx 180 ry 0 rz 180 deg; joints [-53.2, -14.474, 87.043, 77.369, 55.144, -68.59]
  Call Extruder(7.93762)
  MoveL 4696 to (-38.89, 156.67, 78.65) mm, rotated rx 180 ry 0 rz 180 deg; joints [-53.191, -14.517, 87.075, 77.358, 55.138, -68.574]
  MoveL 4697 to (-38.89, 156.67, 78.65) mm, rotated rx 180 ry 0 rz 180 deg; joints [-53.191, -14.517, 87.075, 77.358, 55.138, -68.574]
  Call Extruder(8.09561)
  MoveL 4698 to (-39, 156.42, 78.65) mm, rotated rx -180 ry 0 rz 180 deg; joints [-53.18, -14.554, 87.103, 77.346, 55.13, -68.56]
  MoveL 4699 to (-39, 156.42, 78.65) mm, rotated rx -180 ry 0 rz 180 deg; joints [-53.18, -14.554, 87.103, 77.346, 55.13, -68.56]
  Call Extruder(8.25300)
  MoveL 4700 to (-39.11, 156.17, 78.65) mm, rotated rx 180 ry 0 rz 180 deg; joints [-53.17, -14.591, 87.131, 77.335, 55.122, -68.546]
  MoveL 4701 to (-39.11, 156.17, 78.65) mm, rotated rx 180 ry 0 rz 180 deg; joints [-53.17, -14.591, 87.131, 77.335, 55.122, -68.546]
  Call Extruder(8.43572)
  MoveL 4702 to (-39.22, 155.87, 78.65) mm, rotated rx -180 ry 0 rz 180 deg; joints [-53.156, -14.634, 87.163, 77.322, 55.112, -68.53]
  MoveL 4703 to (-39.22, 155.87, 78.65) mm, rotated rx -180 ry 0 rz 180 deg; joints [-53.156, -14.634, 87.163, 77.322, 55.112, -68.53]
  Call Extruder(8.61768)
  MoveL 4704 to (-39.35, 155.58, 78.65) mm, rotated rx -180 ry 0 rz 180 deg; joints [-53.143, -14.677, 87.195, 77.308, 55.103, -68.513]
  MoveL 4705 to (-39.35, 155.58, 78.65) mm, rotated rx -180 ry 0 rz 180 deg; joints [-53.143, -14.677, 87.195, 77.308, 55.103, -68.513]
  Call Extruder(8.76501)
  MoveL 4706 to (-39.44, 155.34, 78.65) mm, rotated rx 180 ry 0 rz 180 deg; joints [-53.131, -14.712, 87.221, 77.297, 55.093, -68.5]
  MoveL 4707 to (-39.44, 155.34, 78.65) mm, rotated rx 180 ry 0 rz 180 deg; joints [-53.131, -14.712, 87.221, 77.297, 55.093, -68.5]
  Call Extruder(8.87825)
  MoveL 4708 to (-39.5, 155.15, 78.65) mm, rotated rx -180 ry 0 rz 180 deg; joints [-53.121, -14.739, 87.24, 77.288, 55.085, -68.489]
  MoveL 4709 to (-39.5, 155.15, 78.65) mm, rotated rx -180 ry 0 rz 180 deg; joints [-53.121, -14.739, 87.24, 77.288, 55.085, -68.489]
  Call Extruder(8.99103)
  MoveL 4710 to (-39.56, 154.97, 78.65) mm, rotated rx 180 ry 0 rz 180 deg; joints [-53.11, -14.765, 87.26, 77.278, 55.077, -68.478]
  MoveL 4711 to (-39.56, 154.97, 78.65) mm, rotated rx 180 ry 0 rz 180 deg; joints [-53.11, -14.765, 87.26, 77.278, 55.077, -68.478]
  Call Extruder(9.10338)
  MoveL 4712 to (-39.62, 154.78, 78.65) mm, rotated rx -180 ry 0 rz 180 deg; joints [-53.099, -14.792, 87.279, 77.269, 55.068, -68.467]
  MoveL 4713 to (-39.62, 154.78, 78.65) mm, rotated rx -180 ry 0 rz 180 deg; joints [-53.099, -14.792, 87.279, 77.269, 55.068, -68.467]
  Call Extruder(9.21528)
  MoveL 4714 to (-39.68, 154.59, 78.65) mm, rotated rx 180 ry 0 rz -180 deg; joints [-53.088, -14.818, 87.299, 77.259, 55.059, -68.456]
  MoveL 4715 to (-39.68, 154.59, 78.65) mm, rotated rx 180 ry 0 rz -180 deg; joints [-53.088, -14.818, 87.299, 77.259, 55.059, -68.456]
  Call Extruder(9.33668)
  MoveL 4716 to (-39.75, 154.38, 78.65) mm, rotated rx 180 ry 0 rz 180 deg; joints [-53.076, -14.847, 87.32, 77.249, 55.05, -68.444]
  MoveL 4717 to (-39.75, 154.38, 78.65) mm, rotated rx 180 ry 0 rz 180 deg; joints [-53.076, -14.847, 87.32, 77.249, 55.05, -68.444]
  Call Extruder(9.46748)
  MoveL 4718 to (-39.81, 154.16, 78.65) mm, rotated rx 180 ry 0 rz 180 deg; joints [-53.063, -14.878, 87.343, 77.237, 55.039, -68.431]
  MoveL 4719 to (-39.81, 154.16, 78.65) mm, rotated rx 180 ry 0 rz 180 deg; joints [-53.063, -14.878, 87.343, 77.237, 55.039, -68.431]
  Call Extruder(9.59770)
  MoveL 4720 to (-39.88, 153.94, 78.65) mm, rotated rx 180 ry 0 rz 180 deg; joints [-53.049, -14.908, 87.366, 77.225, 55.028, -68.418]
  MoveL 4721 to (-39.88, 153.94, 78.65) mm, rotated rx 180 ry 0 rz 180 deg; joints [-53.049, -14.908, 87.366, 77.225, 55.028, -68.418]
  Call Extruder(9.72737)
  MoveL 4722 to (-39.95, 153.71, 78.65) mm, rotated rx 180 ry 0 rz -180 deg; joints [-53.036, -14.939, 87.389, 77.214, 55.017, -68.405]
  MoveL 4723 to (-39.95, 153.71, 78.65) mm, rotated rx 180 ry 0 rz -180 deg; joints [-53.036, -14.939, 87.389, 77.214, 55.017, -68.405]
  Call Extruder(9.85647)
  MoveL 4724 to (-40.02, 153.49, 78.65) mm, rotated rx -180 ry 0 rz 180 deg; joints [-53.022, -14.97, 87.411, 77.202, 55.007, -68.392]
  MoveL 4725 to (-40.02, 153.49, 78.65) mm, rotated rx -180 ry 0 rz 180 deg; joints [-53.022, -14.97, 87.411, 77.202, 55.007, -68.392]
  Call Extruder(9.97156)
  MoveL 4726 to (-40.06, 153.28, 78.65) mm, rotated rx 180 ry 0 rz 180 deg; joints [-53.007, -14.997, 87.431, 77.191, 54.994, -68.38]
  MoveL 4727 to (-40.06, 153.28, 78.65) mm, rotated rx 180 ry 0 rz 180 deg; joints [-53.007, -14.997, 87.431, 77.191, 54.994, -68.38]
  Call Extruder(10.08619)
  MoveL 4728 to (-40.11, 153.08, 78.65) mm, rotated rx 180 ry 0 rz 180 deg; joints [-52.993, -15.024, 87.451, 77.179, 54.982, -68.367]
  MoveL 4729 to (-40.11, 153.08, 78.65) mm, rotated rx 180 ry 0 rz 180 deg; joints [-52.993, -15.024, 87.451, 77.179, 54.982, -68.367]
  Call Extruder(10.20037)
  MoveL 4730 to (-40.15, 152.88, 78.65) mm, rotated rx -180 ry 0 rz 180 deg; joints [-52.978, -15.05, 87.47, 77.168, 54.97, -68.355]
  MoveL 4731 to (-40.15, 152.88, 78.65) mm, rotated rx -180 ry 0 rz 180 deg; joints [-52.978, -15.05, 87.47, 77.168, 54.97, -68.355]
  Call Extruder(10.31410)
  MoveL 4732 to (-40.2, 152.67, 78.65) mm, rotated rx -180 ry 0 rz 180 deg; joints [-52.963, -15.077, 87.49, 77.156, 54.958, -68.343]
  MoveL 4733 to (-40.2, 152.67, 78.65) mm, rotated rx -180 ry 0 rz 180 deg; joints [-52.963, -15.077, 87.49, 77.156, 54.958, -68.343]
  Call Extruder(10.43953)
  MoveL 4734 to (-40.24, 152.45, 78.65) mm, rotated rx -180 ry 0 rz 180 deg; joints [-52.946, -15.106, 87.512, 77.144, 54.944, -68.329]
  MoveL 4735 to (-40.24, 152.45, 78.65) mm, rotated rx -180 ry 0 rz 180 deg; joints [-52.946, -15.106, 87.512, 77.144, 54.944, -68.329]
  Call Extruder(10.57650)
  MoveL 4736 to (-40.29, 152.2, 78.65) mm, rotated rx 180 ry 0 rz 180 deg; joints [-52.928, -15.138, 87.535, 77.129, 54.929, -68.314]
  MoveL 4737 to (-40.29, 152.2, 78.65) mm, rotated rx 180 ry 0 rz 180 deg; joints [-52.928, -15.138, 87.535, 77.129, 54.929, -68.314]
  Call Extruder(10.71287)
  MoveL 4738 to (-40.34, 151.95, 78.65) mm, rotated rx 180 ry 0 rz 180 deg; joints [-52.909, -15.171, 87.559, 77.115, 54.913, -68.299]
  MoveL 4739 to (-40.34, 151.95, 78.65) mm, rotated rx 180 ry 0 rz 180 deg; joints [-52.909, -15.171, 87.559, 77.115, 54.913, -68.299]
  Call Extruder(10.84862)
